(* IEC 61131-3 sources: elnaProjects/ElpcLogic/PomarKc7Unchanged/build_USO_ecl (part 6) *)

  IF NOT onInit THEN

         fb_kran4Close(phaseNumber:=1, act:=_off);
         fb_kran3bOpen(phaseNumber:=2, act:=_on);
              fb_mvOff(phaseNumber:=3, act:=_off);
              fb_pnsOn(phaseNumber:=4, act:=_on);
         fb_kran1Close(phaseNumber:=6, act:=_off);
         fb_kran2Close(phaseNumber:=7, act:=_off);
          fb_kran5Open(phaseNumber:=8, act:=_on);
          fb_autoNuOff(phaseNumber:=9, act:=_reset, waitCompletion:=FALSE);
         fb_autoPnsOff(phaseNumber:=10, act:=_reset, waitCompletion:=FALSE);
        fb_autoAvomOff(phaseNumber:=11, act:=_reset, waitCompletion:=FALSE);
        fb_avom1cmdOff(phaseNumber:=12, act:=_off);
        fb_avom2cmdOff(phaseNumber:=13, act:=_off);
      fb_pInNagLess100(phaseNumber:=14);
           fb_waitKran(phaseNumber:=15, delay:=T#240S);
         fb_pnsWaitOff(phaseNumber:=17, act:=_run, waitCompletion:=TRUE);
             fb_nu1off(phaseNumber:=18, act:=_off);
             fb_nu2off(phaseNumber:=19, act:=_off);
    fb_runUnsuccessful(phaseNumber:=20);

  onInit:=TRUE;
  END_IF;

         fb_kran4Close(StrPh:=kran4Close, Im:=Im.kran4);
         fb_kran3bOpen(StrPh:=kran3bOpen, Im:=Im.kran3b);
              fb_mvOff(StrPh:=mvOff, Im:=Im.mv);
              fb_pnsOn(StrPh:=pnsOn, Im:=Im.pns);

         fb_kran1Close(StrPh:=kran1Close, Im:=Im.kran1);
         fb_kran2Close(StrPh:=kran2Close, Im:=Im.kran2);
          fb_kran5Open(StrPh:=kran5Open, Im:=Im.kran5);
          fb_autoNuOff(StrPh:=autoNuOff, alg:=algoritms.autoNu);
         fb_autoPnsOff(StrPh:=autoPnsOff, alg:=algoritms.autoPns);
        fb_autoAvomOff(StrPh:=autoAvomOff, alg:=algoritms.AutoAvom);
        fb_avom1cmdOff(StrPh:=avom1cmdOff, Im:=Im.v1_Avom);
        fb_avom2cmdOff(StrPh:=avom2cmdOff, Im:=Im.v2_Avom);
      fb_pInNagLess100(StrPh:=pInNagLess100);
           fb_waitKran(StrPh:=waitKran, timer:=AlgTimers.AO_waitKran);
         fb_pnsWaitOff(StrPh:=pnsWaitOff, alg:=algoritms.vibegPNS, waitCompletion:=TRUE);
             fb_nu1off(StrPh:=nu1off, Im:=Im.nu1);
             fb_nu2off(StrPh:=nu2off, Im:=Im.nu2);
    fb_runUnsuccessful(StrPh:=runUnsuccessful);

  StrAlg.CanRun := StrAlg.inCanRun;
  StrAlg.OpcCommandsDisabled := StrAlg.inOpcCommandsDisabled;

  IF StrAlg.isRuning THEN

      StrAlg.hasError := kran4Close.error OR mvOff.error OR pnsOn.error OR kran3bOpen.error
      OR kran1Close.error OR kran2Close.error OR kran5Open.error OR runUnsuccessful.error;

      runPhase(kran4Close);
      runPhase(kran3bOpen);
      runPhase(kran1Close);
      runPhase(kran2Close);
      runPhase(mvOff);

      IF kran1Close.top AND kran2Close.top AND kran4Close.top THEN
          runPhase(kran5Open);
      END_IF;

      IF mvOff.top THEN
            runPhase(autoPnsOff);
      END_IF;

       IF autoPnsOff.top THEN
  	runPhase(pnsOn);
      END_IF;

      IF kran5Open.top THEN
         runPhase(pInNagLess100);
         resetPhase(waitKran);
      END_IF;

     IF pInNagLess100.start AND NOT pInNagLess100.top THEN
  	pInNagLess100.top:=( ai.P_gaza_na_vkhode_nagnetatelia.interval >= _statusAi.NORMAL AND
            ai.P_gaza_na_vkhode_nagnetatelia.value < Ust_Pgaza ) AND
           (ai.P_gaza_na_vykhode_nagnetatelia.interval >= _statusAi.NORMAL AND
            ai.P_gaza_na_vykhode_nagnetatelia.value < Ust_Pgaza);

     END_IF;

      IF pInNagLess100.top AND kran3bOpen.top AND mvOff.top THEN
  	ai.dPmaslo_gaz.Disabled_LA:=TRUE;
            ai.dPmaslo_gaz.Disabled_LW:=TRUE;
            IM.SingleSignals.dP_oilgaz_low.Disabled_Sig:=TRUE;
            resetAiProtection(protections.dP_maslogaz_LA);
            resetDiProtection(protections.dP_masloGaz_LowDI);

            runPhase(autoNuOff);
            runPhase(nu1off);
            runPhase(nu2off);
      END_IF;

       IF nu1off.top AND  nu2off.top THEN
  	runPhase(pnsWaitOff);
      END_IF;

      IF waitKran.top AND (NOT kran5Open.top) THEN
  	runUnsuccessful.error:=TRUE;
      END_IF;

      IF pnsWaitOff.top THEN
  	runPhase(autoAvomOff);
      END_IF;

      IF autoAvomOff.top THEN
  	runPhase(avom1cmdOff);
  	runPhase(avom2cmdOff);
      END_IF;

      IF avom1cmdOff.top AND avom2cmdOff.top THEN
  	 StrAlg.opcCommandsDisabled:=FALSE;
      END_IF;

      StrAlg.isEnded:= avom1cmdOff.top AND avom2cmdOff.top;
  END_IF;

  StrAlg.CanRun := StrAlg.inCanRun;
  StrAlg.OpcCommandsDisabled := StrAlg.inOpcCommandsDisabled;

  (* ---- Если управление с ВУ заблокировано, то  передаем команду из алгоритма ---- *)
  IF StrAlg.inOpcCommandsDisabled THEN
  	StrAlg.inCommand := StrAlg.inCommand_Alg;
  ELSE (* иначе передаем команду с АРМа*)
  	StrAlg.inCommand := StrAlg.inCommand_ARM;
  END_IF;

  _sunpackerCommand(command := StrAlg.inCommand);
  	source := _sunpackerCommand.source;
  	cmd := _sunpackerCommand.cmd;

  IF cmd <> 0 AND lastCmd <> cmd AND (((NOT StrAlg.opcCommandsDisabled) AND source > 0) OR source = 0) then
  	CASE BYTE_TO_INT(cmd) OF
  		(*cmdRun*) 1: 	IF (StrAlg.CanRun) THEN
  					StrAlg.isRuning := TRUE;
  					StrAlg.isEnded := FALSE;
  					StrAlg.hasError := FALSE;
  					(*****************       OnRun       *****************)

                                                    StrAlg.opcCommandsDisabled:=TRUE;
                                                    runIfNotRunningSO(IM.SingleOutputs.IndikicijaAS_fonar);
                                                    runIfNotRunningSO(IM.SingleOutputs.AO_GPA);
                                                    stopPusk(algoritms);
                                                    algManager.nMode:=ModeGpa.MODE_AO;

                                                    runPhase(waitKran);
                                                    runPhase(runUnsuccessful);

                                                    resetDiProtection(protections.mvOff);
                                                    resetAiProtection(protections.Vibratciia_rotora_nagnetatelia_t1_HA);
                                                    resetAiProtection(protections.Vibratciia_rotora_nagnetatelia_t2_HA);
                                                    resetAiProtection(protections.Vibratciia_rotora_nagnetatelia_t3_HA);
                                                    resetAiProtection(protections.Vibratciia_rotora_nagnetatelia_t4_HA);
                                                    resetAiProtection(protections.Vibratciia_STD_t1_HA);
                                                    resetAiProtection(protections.Vibratciia_STD_t2_HA);
                                                    resetDiProtection(protections.Kran1sdvig);
                                                    resetDiProtection(protections.Kran2sdvig);

  					cmd_for_Status := cmd;
  					source_for_Status := source;
  					command_error_for_Status := 0;
  				ELSE
  					StrAlg.isRuning := FALSE;
  					StrAlg.isEnded := FALSE;
  					StrAlg.hasError 	:= FALSE;

  					cmd_for_Status := 0;
  					source_for_Status := source;
  					command_error_for_Status := cmd;
  				END_IF;
  		(*cmdReset*) 2: 	StrAlg.isRuning := FALSE;
  				StrAlg.isEnded := FALSE;
  				StrAlg.hasError 	:= FALSE;

                                           (*****************       OnReset       *****************)
                                          protectManager.inCommand:=PMcommand.RestartAllSignaling;
                                          waitReset(IN:=FALSE);
                                          resetIfRunningSO(IM.SingleOutputs.IndikicijaAS_fonar);
                                          resetIfRunningSO(IM.SingleOutputs.AO_GPA);
                                          resetIfRunning(algoritms.vibegPNS);
                                          algManager.nMode:=ModeGpa.MODE_STOP;
                                          impulseSO(Im.SingleOutputs.SbrosBREO);

                                          resetPhase(kran4Close);
                                          resetPhase(mvOff);
                                          resetPhase(pnsOn);
                                          resetPhase(kran3bOpen);
                                          resetPhase(kran1Close);
                                          resetPhase(kran2Close);
                                          resetPhase(kran5Open);
                                          resetPhase(autoNuOff);
                                          resetPhase(autoPnsOff);
                                          resetPhase(pInNagLess100);
  	                              resetPhase(autoAvomOff);
                                          resetPhase(avom1cmdOff);
                                          resetPhase(avom2cmdOff);
                                          resetPhase(nu1off);
                                          resetPhase(nu2off);
                                          resetPhase(waitKran);
                                          resetPhase(pnsWaitOff);
                                          resetPhase(runUnsuccessful);

  				cmd_for_Status := cmd;
  				source_for_Status := source;
  				command_error_for_Status := 0;
  	END_CASE;
  	resetCmdTimer(IN := false);
  	resetCmdTimerPriznak := TRUE;
  END_IF;
  lastCmd := cmd;

  resetCmdTimer(IN := resetCmdTimerPriznak, PT := T#5S);
  IF resetCmdTimer.Q THEN
  	resetCmdTimerPriznak := FALSE;
  	source_for_Status := 0;
  	cmd_for_Status := 0;
  	command_error_for_Status := 0;
  END_IF;

  StrAlg.Start:= kran4Close.startStatus
              OR mvOff.startStatus
              OR pnsOn.startStatus
              OR kran3bOpen.startStatus
              OR kran1Close.startStatus
              OR kran2Close.startStatus
              OR kran5Open.startStatus
              OR autoNuOff.startStatus
              OR autoPnsOff.startStatus
              OR pInNagLess100.startStatus
              OR autoAvomOff.startStatus
              OR avom1cmdOff.startStatus
              OR avom2cmdOff.startStatus
              OR nu1off.startStatus
              OR nu2off.startStatus
              OR waitKran.startStatus
              OR pnsWaitOff.startStatus
              OR runUnsuccessful.startStatus;

  StrAlg.Error:= kran4Close.errorStatus
              OR mvOff.errorStatus
              OR pnsOn.errorStatus
              OR kran3bOpen.errorStatus
              OR kran1Close.errorStatus
              OR kran2Close.errorStatus
              OR kran5Open.errorStatus
              OR autoNuOff.errorStatus
              OR autoPnsOff.errorStatus
              OR pInNagLess100.errorStatus
              OR autoAvomOff.errorStatus
              OR avom1cmdOff.errorStatus
              OR avom2cmdOff.errorStatus
              OR nu1off.errorStatus
              OR nu2off.errorStatus
              OR waitKran.errorStatus
              OR pnsWaitOff.errorStatus
              OR runUnsuccessful.errorStatus;

  StrAlg.Top:=   kran4Close.topStatus
              OR mvOff.topStatus
              OR pnsOn.topStatus
              OR kran3bOpen.topStatus
              OR kran1Close.topStatus
              OR kran2Close.topStatus
              OR kran5Open.topStatus
              OR autoNuOff.topStatus
              OR autoPnsOff.topStatus
              OR pInNagLess100.topStatus
              OR autoAvomOff.topStatus
              OR avom1cmdOff.topStatus
              OR avom2cmdOff.topStatus
              OR nu1off.topStatus
              OR nu2off.topStatus
              OR waitKran.topStatus
              OR pnsWaitOff.topStatus
              OR runUnsuccessful.topStatus;

  (*TODO: TYPE PROGRAM CODE HERE*)
  StrAlg.status :=  SHL(BYTE_TO_DWORD(source_for_Status), 29)
  			OR SHL(BYTE_TO_DWORD(cmd_for_Status), 26)
  			OR SHL(BYTE_TO_DWORD(command_error_for_Status), 23)
  			OR SHL(BOOL_TO_DWORD(StrAlg.OpcCommandsDisabled ), 21)
  			OR SHL(BOOL_TO_DWORD(StrAlg.hasError),4)
  			OR SHL(BOOL_TO_DWORD(StrAlg.CanRun),2)
  			OR SHL(BOOL_TO_DWORD(StrAlg.isEnded),1)
  			OR BOOL_TO_DWORD(StrAlg.isRuning);
END_FUNCTION_BLOCK

FUNCTION NapryageniaOK : BOOL
  VAR_INPUT
    im : ImConfig;
  END_VAR

  NapryageniaOK:=
  NOT (Im.SingleSignals.NS_G1_G2.Q
  OR Im.SingleSignals.NS_G10_G11.Q
  OR Im.SingleSignals.NS_G13_G14.Q
  OR Im.SingleSignals.NS_G15_G16.Q
  OR Im.SingleSignals.NS_G17.Q
  OR Im.SingleSignals.NS_G18_G19.Q
  OR Im.SingleSignals.NS_G3_G4.Q
  OR Im.SingleSignals.NS_G5_G6.Q
  OR Im.SingleSignals.NS_G7_G8.Q
  OR im.SingleSignals.QF1_on.Q
  OR Im.SingleSignals.QF2_on.Q
  OR Im.SingleSignals.QF23_on.Q
  OR Im.SingleSignals.QF4_QF5_on.Q
  OR Im.SingleSignals.QF6_QF7_on.Q
  OR Im.SingleSignals.QF8_QF9_on.Q
  OR Im.SingleSignals.QF10_QF11_on.Q
  OR im.SingleSignals.QF12_QF13_on.Q
  OR im.SingleSignals.QF22_on.Q
  OR Im.SingleSignals.QF14_QF15_on.Q);
END_FUNCTION

FUNCTION nsCepeiUpravlenya : BOOL
  VAR_INPUT
    im : ImConfig;
  END_VAR

  nsCepeiUpravlenya:=
  	im.kran1.So OR im.kran1.Sz OR
  	im.kran2.So OR im.kran2.Sz OR
  	im.kran4.So OR im.kran4.Sz OR
  	im.kran5.So OR im.kran5.Sz OR
  	(*im.kran6.So OR im.kran6.Sz OR*)
  	im.kran3b.So OR im.kran3b.Sz OR
  	im.pns.breakCmdOn OR
  	im.nu1.breakCmdOn OR
  	im.nu2.breakCmdOn OR
  	im.PNS.breakCmdOn OR
            im.v1_Avom.breakCmdOn OR
            im.v2_Avom.breakCmdOn OR
            (*im.Ten.breakCmdOn OR*)
  	im.mv.breakCmdOff;
END_FUNCTION

FUNCTION discretNS : BOOL
  VAR_INPUT
    di : DiConfig;
  END_VAR

  discretNS:=  ((di.di_0.reliability <> 255)
                OR (di.di_1.reliability <> 255)
                OR (di.di_2.reliability <> 255)
                OR (di.di_3.reliability <> 255)
                OR (di.di_4.reliability <> 255)
                OR (di.di_5.reliability <> 255)
                OR (di.di_6.reliability <> 255)
                OR (di.di_7.reliability <> 255)
                OR (di.di_8.reliability <> 255)
                OR (di.di_9.reliability <> 255)
                OR (di.di_10.reliability <> 255)
                OR (di.di_11.reliability <> 255)
                OR (di.di_12.reliability <> 255)
                OR (di.di_13.reliability <> 255)
                OR (di.di_14.reliability <> 255));
               (* OR (di.di_15.reliability <> 255)); *)
END_FUNCTION

FUNCTION analogsNS : BOOL
  VAR_INPUT
    ai : AiConfig;
  END_VAR
  VAR
    statusAi : TYPE_StatusAi;
  END_VAR

  analogsNS:=
    ((ai.T_obmotki_fazy_1_k.Interval < statusAi.Normal) AND NOT ai.T_obmotki_fazy_1_k.remont)
  OR((ai.T_aktivnogo_zheleza_statora_1_k.Interval < statusAi.Normal) AND NOT ai.T_aktivnogo_zheleza_statora_1_k.remont)
  OR((ai.T_obmotki_fazy_2_k.Interval < statusAi.Normal) AND NOT ai.T_obmotki_fazy_2_k.remont)
  OR((ai.T_aktivnogo_zheleza_statora_2_k.Interval < statusAi.Normal) AND NOT ai.T_aktivnogo_zheleza_statora_2_k.remont)
  OR((ai.T_obmotki_fazy_3_k.Interval < statusAi.Normal) AND NOT ai.T_obmotki_fazy_3_k.remont)
  OR((ai.T_aktivnogo_zheleza_statora_3_k.Interval < statusAi.Normal) AND NOT ai.T_aktivnogo_zheleza_statora_3_k.remont)
  OR((ai.T_masla_v_maslobake.Interval < statusAi.Normal) AND NOT ai.T_masla_v_maslobake.remont)
  OR((ai.T_perednego_opornogo_podshipnika_dvigatelia_t1.Interval < statusAi.Normal) AND NOT ai.T_perednego_opornogo_podshipnika_dvigatelia_t1.remont)
  OR((ai.T_zadnego_opornogo_podshipnika_dvigatelia_t2.Interval < statusAi.Normal) AND NOT ai.T_zadnego_opornogo_podshipnika_dvigatelia_t2.remont)
  OR((ai.T_masla_na_slive_perednego_opornogo_podshipnika_dvigatelia.Interval < statusAi.Normal) AND NOT ai.T_masla_na_slive_perednego_opornogo_podshipnika_dvigatelia.remont)
  OR((ai.T_masla_na_slive_zadnego_opornogo_podshipnika_dvigatelia.Interval < statusAi.Normal) AND NOT ai.T_masla_na_slive_zadnego_opornogo_podshipnika_dvigatelia.remont)
  OR((ai.T_podshipnika_reduktora_t1.Interval < statusAi.Normal) AND NOT ai.T_podshipnika_reduktora_t1.remont)
  OR((ai.T_podshipnika_reduktora_t2.Interval < statusAi.Normal) AND NOT ai.T_podshipnika_reduktora_t2.remont)
  OR((ai.T_podshipnika_reduktora_t3.Interval < statusAi.Normal) AND NOT ai.T_podshipnika_reduktora_t3.remont)
  OR((ai.T_podshipnika_reduktora_t4.Interval < statusAi.Normal) AND NOT ai.T_podshipnika_reduktora_t4.remont)
  OR((ai.T_opornogo_podshipnika_nagnetatelia_t1.Interval < statusAi.Normal) AND NOT ai.T_opornogo_podshipnika_nagnetatelia_t1.remont)
  OR((ai.T_opornogo_podshipnika_nagnetatelia_t2.Interval < statusAi.Normal) AND NOT ai.T_opornogo_podshipnika_nagnetatelia_t2.remont)
  OR((ai.T_opornogo_podshipnika_nagnetatelia_t3.Interval < statusAi.Normal) AND NOT ai.T_opornogo_podshipnika_nagnetatelia_t3.remont)
  OR((ai.T_oporno_upornogo_podshipnika_nagnetatelia_t4.Interval < statusAi.Normal) AND NOT ai.T_oporno_upornogo_podshipnika_nagnetatelia_t4.remont)
  OR((ai.T_masla_do_AVOM.Interval < statusAi.Normal) AND NOT ai.T_masla_do_AVOM.remont)
  OR((ai.T_masla_posle_AVOM.Interval < statusAi.Normal) AND NOT ai.T_masla_posle_AVOM.remont)
  OR((ai.T_gaz_in_nagnetatelia.Interval < statusAi.Normal) AND NOT ai.T_gaz_in_nagnetatelia.remont)
  OR((ai.T_gaz_out_nagnetatelia.Interval < statusAi.Normal) AND NOT ai.T_gaz_out_nagnetatelia.remont)
  OR((ai.T_clodAir_dvigatelia_t1.Interval < statusAi.Normal) AND NOT ai.T_clodAir_dvigatelia_t1.remont)
  OR((ai.T_hotAir_dvigatelia_t1.Interval < statusAi.Normal) AND NOT ai.T_hotAir_dvigatelia_t1.remont)
  OR((ai.dPmaslo_gaz.Interval < statusAi.Normal) AND NOT ai.dPmaslo_gaz.remont)
  OR((ai.dP_gaza_na_konfuzore_nagnetatelia.Interval < statusAi.Normal) AND NOT ai.dP_gaza_na_konfuzore_nagnetatelia.remont)
  OR((ai.P_masla_uplotneniia.Interval < statusAi.Normal) AND NOT ai.P_masla_uplotneniia.remont)
  OR((ai.P_gaza_na_vkhode_nagnetatelia.Interval < statusAi.Normal) AND NOT ai.P_gaza_na_vkhode_nagnetatelia.remont)
  OR((ai.P_gaza_na_vykhode_nagnetatelia.Interval < statusAi.Normal) AND NOT ai.P_gaza_na_vykhode_nagnetatelia.remont)
  OR((ai.P_masla_smazki_nizkoe.Interval < statusAi.Normal) AND NOT ai.P_masla_smazki_nizkoe.remont)
  OR((ai.P_masla_smazki_srednee_posle_nasosov.Interval < statusAi.Normal) AND NOT ai.P_masla_smazki_srednee_posle_nasosov.remont)
  OR((ai.Vibratciia_STD_t1.Interval < statusAi.Normal) AND NOT ai.Vibratciia_STD_t1.remont)
  OR((ai.Vibratciia_STD_t2.Interval < statusAi.Normal) AND NOT ai.Vibratciia_STD_t2.remont)
  OR((ai.Vibratciia_rotora_nagnetatelia_t1.Interval < statusAi.Normal) AND NOT ai.Vibratciia_rotora_nagnetatelia_t1.remont)
  OR((ai.Vibratciia_rotora_nagnetatelia_t2.Interval < statusAi.Normal) AND NOT ai.Vibratciia_rotora_nagnetatelia_t2.remont)
  OR((ai.Vibratciia_rotora_nagnetatelia_t3.Interval < statusAi.Normal) AND NOT ai.Vibratciia_rotora_nagnetatelia_t3.remont)
  OR((ai.Vibratciia_rotora_nagnetatelia_t4.Interval < statusAi.Normal) AND NOT ai.Vibratciia_rotora_nagnetatelia_t4.remont)
  OR((ai.Osevoi_sdvig_rotora_nagnetatelia.Interval < statusAi.Normal) AND NOT ai.Osevoi_sdvig_rotora_nagnetatelia.remont)
  OR((ai.Uroven_masla_v_maslobake.Interval < statusAi.Normal) AND NOT ai.Uroven_masla_v_maslobake.remont)
  OR((ai.Tok_vozbuzhdeniia_vozbuditelia.Interval < statusAi.Normal) AND NOT ai.Tok_vozbuzhdeniia_vozbuditelia.remont)
  OR((ai.Tok_statora_elektrodvigatelia.Interval < statusAi.Normal) AND NOT ai.Tok_statora_elektrodvigatelia.remont)
  OR((ai.Aktivnaia_moshchnost.Interval < statusAi.Normal) AND NOT ai.Aktivnaia_moshchnost.remont)
  OR((ai.Reaktivnaia_moshchnost.Interval < statusAi.Normal) AND NOT ai.Reaktivnaia_moshchnost.remont)
  OR((ai.VoltageSHU_osnovnoi_vvod.Interval < statusAi.Normal) AND NOT ai.VoltageSHU_osnovnoi_vvod.remont)
  OR((ai.VoltageSHU_rezervnyi_vvod.Interval < statusAi.Normal) AND NOT ai.VoltageSHU_rezervnyi_vvod.remont);
END_FUNCTION

FUNCTION nsCepeiControl : BOOL
  VAR_INPUT
    im : ImConfig;
  END_VAR

  nsCepeiControl:= NOT (
  	im.kran1.reliability OR
  	im.kran2.reliability OR
  	im.kran4.reliability OR
  	im.kran5.reliability OR
  	im.kran6.reliability OR
  	im.kran3b.reliability OR
  	im.pns.reliability OR
  	im.nu1.reliability OR
  	im.nu2.reliability OR
  	im.PNS.reliability OR
            im.v1_Avom.reliability OR
            im.v2_Avom.reliability OR
            im.Ten.reliability OR
  	im.mv.reliability);
END_FUNCTION

FUNCTION_BLOCK ppuAlg
  VAR_IN_OUT
    StrAlg : struct_Alg;
  END_VAR
  VAR
    Sau_ok : struct_PhaseAlgoritm;
    Voltage_ok : struct_PhaseAlgoritm;
    controlCircuits_ok : struct_PhaseAlgoritm;
    controlCircuitsIM_ok : struct_PhaseAlgoritm;
  END_VAR
  VAR_IN_OUT
    BEAO_otKnSHU : struct_PhaseAlgoritm;
    circuitAO_ok : struct_PhaseAlgoritm;
    BREO_Srabotal : struct_PhaseAlgoritm;
    DI_ok : struct_PhaseAlgoritm;
    AI_ok : struct_PhaseAlgoritm;
    Loil_ok : struct_PhaseAlgoritm;
    Toil_ok : struct_PhaseAlgoritm;
    mvOff : struct_PhaseAlgoritm;
    Kr_1_close : struct_PhaseAlgoritm;
    Kr_2_close : struct_PhaseAlgoritm;
    Kr_3b_open : struct_PhaseAlgoritm;
    Kr_4_close : struct_PhaseAlgoritm;
    Kr_5_open : struct_PhaseAlgoritm;
    PNS_off : struct_PhaseAlgoritm;
    NU_1_off : struct_PhaseAlgoritm;
    NU_2_off : struct_PhaseAlgoritm;
    Avom_1_off : struct_PhaseAlgoritm;
    Avom_2_off : struct_PhaseAlgoritm;
    Est_rezerv_NU : struct_PhaseAlgoritm;
    Not_AO_NO_EAO : struct_PhaseAlgoritm;
    Not_AS_PS : struct_PhaseAlgoritm;
    BusketTest : struct_PhaseAlgoritm;
    BusketRolledIn : struct_PhaseAlgoritm;
  END_VAR
  VAR
    fb_Sau_ok : fb_ph_CustomPhase;
    fb_Voltage_ok : fb_ph_CustomPhase;
    fb_controlCircuits_ok : fb_ph_CustomPhase;
    fb_controlCircuitsIM_ok : fb_ph_CustomPhase;
    fb_BEAO_otKnSHU : fb_ph_CustomPhase;
    fb_circuitAO_ok : fb_ph_CustomPhase;
    fb_BREO_Srabotal : fb_ph_CustomPhase;
    fb_DI_ok : fb_ph_CustomPhase;
    fb_AI_ok : fb_ph_CustomPhase;
    fb_Loil_ok : fb_ph_CustomPhase;
    fb_Toil_ok : fb_ph_CustomPhase;
    fb_mvOff : fb_ph_CustomPhase;
    fb_Kr_1_close : fb_ph_CustomPhase;
    fb_Kr_2_close : fb_ph_CustomPhase;
    fb_Kr_3b_open : fb_ph_CustomPhase;
    fb_Kr_4_close : fb_ph_CustomPhase;
    fb_Kr_5_open : fb_ph_CustomPhase;
    fb_PNS_off : fb_ph_CustomPhase;
    fb_NU_1_off : fb_ph_CustomPhase;
    fb_NU_2_off : fb_ph_CustomPhase;
    fb_Avom_1_off : fb_ph_CustomPhase;
    fb_Avom_2_off : fb_ph_CustomPhase;
    fb_Est_rezerv_NU : fb_ph_CustomPhase;
    fb_Not_AO_NO_EAO : fb_ph_CustomPhase;
    fb_Not_AS_PS : fb_ph_CustomPhase;
    fb_BusketTest : fb_ph_CustomPhase;
    fb_BusketRolledIn : fb_ph_CustomPhase;
    _sunpackerCommand : fb_sunpackerCommand;
    modeR_Trig : R_TRIG;
    modeF_Trig : F_TRIG;
    _statusAi : TYPE_StatusAi;
    _Answers : TYPE_Answers;
    _statusDualInput : TYPE_statusDualInput;
    _DualStateImAction : TYPE_DualStateImAction;
    _PhaseAlgoritmAction : TYPE_PhaseAlgoritmAction;
    _basketStats : TYPE_basketStats;
  END_VAR
  VAR_OUTPUT
    puskAllowed : BOOL;
    testAllowed : BOOL;
  END_VAR
  VAR
    ppuDone : BOOL;
    source : BYTE;
    cmd : BYTE;
    lastCmd : BYTE;
    source_for_Status : BYTE;
    cmd_for_Status : BYTE;
    command_error_for_Status : BYTE;
    resetCmdTimer : TON;
    resetCmdTimerPriznak : BOOL;
    onInit : BOOL;
  END_VAR
  VAR_EXTERNAL
    IM : ImConfig;
    ai : AiConfig;
    di : DiConfig;
    algManager : struct_AlgoritmsManager;
    protectManager : struct_ProtectionsManager;
    NotHasRezervNU : BOOL;
    ModeGpa : TYPE_ModeGpa;
    algoritms : AlgoritmsConfig;
  END_VAR

  IF NOT onInit THEN
                fb_Sau_ok(phaseNumber:=0);
            fb_Voltage_ok(phaseNumber:=1);
    fb_controlCircuits_ok(phaseNumber:=2);
  fb_controlCircuitsIM_ok(phaseNumber:=5);
          fb_BEAO_otKnSHU(phaseNumber:=6);
          fb_circuitAO_ok(phaseNumber:=7);
         fb_BREO_Srabotal(phaseNumber:=9);
                 fb_DI_ok(phaseNumber:=10);
                 fb_AI_ok(phaseNumber:=11);
               fb_Loil_ok(phaseNumber:=12);
               fb_Toil_ok(phaseNumber:=13);
                 fb_mvOff(phaseNumber:=14);
            fb_Kr_1_close(phaseNumber:=15);
            fb_Kr_2_close(phaseNumber:=16);
            fb_Kr_3b_open(phaseNumber:=17);
            fb_Kr_4_close(phaseNumber:=18);
             fb_Kr_5_open(phaseNumber:=19);
               fb_PNS_off(phaseNumber:=20);
              fb_NU_1_off(phaseNumber:=21);
              fb_NU_2_off(phaseNumber:=22);
            fb_Avom_1_off(phaseNumber:=23);
            fb_Avom_2_off(phaseNumber:=24);
         fb_Est_rezerv_NU(phaseNumber:=25);
         fb_Not_AO_NO_EAO(phaseNumber:=26);
             fb_Not_AS_PS(phaseNumber:=27);
            fb_BusketTest(phaseNumber:=28);
        fb_BusketRolledIn(phaseNumber:=29);

  onInit:=TRUE;
  END_IF;

                fb_Sau_ok(StrPh:=Sau_ok);
            fb_Voltage_ok(StrPh:=Voltage_ok);
    fb_controlCircuits_ok(StrPh:=controlCircuits_ok);
  fb_controlCircuitsIM_ok(StrPh:=controlCircuitsIM_ok);
          fb_BEAO_otKnSHU(StrPh:=BEAO_otKnSHU);
          fb_circuitAO_ok(StrPh:=circuitAO_ok);
         fb_BREO_Srabotal(StrPh:=BREO_Srabotal);
                 fb_DI_ok(StrPh:=DI_ok);
                 fb_AI_ok(StrPh:=AI_ok);
               fb_Loil_ok(StrPh:=Loil_ok);
               fb_Toil_ok(StrPh:=Toil_ok);
                 fb_mvOff(StrPh:=mvOff);
            fb_Kr_1_close(StrPh:=Kr_1_close);
            fb_Kr_2_close(StrPh:=Kr_2_close);
            fb_Kr_3b_open(StrPh:=Kr_3b_open);
            fb_Kr_4_close(StrPh:=Kr_4_close);
             fb_Kr_5_open(StrPh:=Kr_5_open);
               fb_PNS_off(StrPh:=PNS_off);
              fb_NU_1_off(StrPh:=NU_1_off);
              fb_NU_2_off(StrPh:=NU_2_off);
            fb_Avom_1_off(StrPh:=Avom_1_off);
            fb_Avom_2_off(StrPh:=Avom_2_off);
         fb_Est_rezerv_NU(StrPh:=Est_rezerv_NU);
         fb_Not_AO_NO_EAO(StrPh:=Not_AO_NO_EAO);
             fb_Not_AS_PS(StrPh:=Not_AS_PS);
            fb_BusketTest(StrPh:=BusketTest);
        fb_BusketRolledIn(StrPh:=BusketRolledIn);

  IF StrAlg.isRuning THEN

      Sau_ok.top:= (*(NOT kontroller.diagnostic.ns)  OR kontroller.imit;*) TRUE;
      Voltage_ok.top	:=NapryageniaOK(IM);
      controlCircuits_ok.top	:=NOT nsCepeiUpravlenya(IM);
      controlCircuitsIM_ok.top	:=NOT nsCepeiControl(IM);
      BEAO_otKnSHU.top	:=NOT Im.singleSignals.BEO_ON_knopkaSHU.Q AND Im.singleSignals.BEO_ON_knopkaSHU.reliability;
      circuitAO_ok.top	:=NOT Im.singleSignals.AO_KC.Q AND Im.singleSignals.AO_KC.reliability;
      BREO_Srabotal.top	:=NOT Im.singleSignals.BEO_Srabat.Q AND Im.singleSignals.BEO_Srabat.reliability;
      DI_ok.top	:=NOT discretNS(di);
      AI_ok.top	:=NOT analogsNS(ai);
      mvOff.top:=Im.mv.onStatus = _statusDualInput.STATUS_OFF;
      Toil_ok.top:=(ai.T_masla_v_maslobake.interval = _statusAi.normal);
      Loil_ok.top:=(ai.Uroven_masla_v_maslobake.interval= _statusAi.normal) ;

      Kr_1_close.top:=Im.kran1.onStatus = _statusDualInput.STATUS_OFF;
      Kr_2_close.top:=Im.kran2.onStatus = _statusDualInput.STATUS_OFF;
      Kr_3b_open.top:=Im.kran3b.onStatus = _statusDualInput.STATUS_ON;
      Kr_4_close.top:=Im.kran4.onStatus = _statusDualInput.STATUS_OFF;
      Kr_5_open.top:=	Im.kran5.onStatus = _statusDualInput.STATUS_ON;
      PNS_off.top:=	Im.pns.onStatus = _statusDualInput.STATUS_OFF;
      NU_1_off.top:=	Im.nu1.onStatus = _statusDualInput.STATUS_OFF;
      NU_2_off.top:=	Im.nu2.onStatus = _statusDualInput.STATUS_OFF;
      Avom_1_off.top:=Im.v1_Avom.onStatus = _statusDualInput.STATUS_OFF;
      Avom_2_off.top:=Im.v2_Avom.onStatus = _statusDualInput.STATUS_OFF;

      Est_rezerv_NU.top:= NOT NotHasRezervNU;
      Not_AO_NO_EAO.top:=	   NOT ( Im.singleOutputs.AO_GPA.q
                                      OR Im.singleSignals.AO_KC.q
                                      OR Im.singleSignals.AOGPA_knopkaSHU.q
                                      OR Im.singleSignals.AOGPA_PRU.q
                                      OR Im.singleSignals.NOGPA_knopkaSHU.q
                                      OR Im.singleSignals.BEO_Srabat.q);

      Not_AS_PS.top:=	NOT (algManager.DiscretPS OR algManager.analogsPS OR algManager.ProtectionSignaling);
      BusketTest.top:=Im.mv.basketStatus = _basketStats.BASKET_ROLLEDOUT;
      BusketRolledIn.top:=Im.mv.basketStatus = _basketStats.BASKET_RolledIN;

      ppuDone:=                 Sau_ok.top AND
  			Voltage_ok.top AND
  			controlCircuits_ok.top AND
  			controlCircuitsIM_ok.top AND
  			circuitAO_ok.top AND
  			BEAO_otKnSHU.top	AND
  			BREO_Srabotal.top	AND
  			DI_ok.top AND
  			AI_ok.top AND
  			Loil_ok.top AND
  			Toil_ok.top AND
  			mvOff.top AND
  			Kr_1_close.top AND
  			Kr_2_close.top AND
  			Kr_3b_open.top AND
  			Kr_4_close.top AND
  			Kr_5_open.top AND
  			PNS_off.top AND
  			NU_1_off.top AND
  			NU_2_off.top AND
  			Avom_1_off.top AND
  			Avom_2_off.top AND
  			Est_rezerv_NU.top AND
  			Not_AO_NO_EAO.top AND
  			Not_AS_PS.top ;

      puskAllowed:= ppuDone AND Im.mv.basketStatus = _basketStats.BASKET_ROLLEDIN;
      testAllowed:= ppuDone AND Im.mv.basketStatus = _basketStats.BASKET_ROLLEDOUT;

      modeR_Trig(CLK:=puskAllowed);
      modeF_Trig(CLK:=puskAllowed);

      IF modeR_Trig.Q THEN
  	algManager.nMode:= ModeGpa.MODE_READY;
      END_IF;
      IF modeF_Trig.Q THEN
  	algManager.nMode:= ModeGpa.MODE_STOP;
      END_IF;

      IF puskAllowed THEN
          algoritms.Apusk.inCanRun:= TRUE;
          algoritms.SemiAutoPusk.inCanRun:= TRUE;
      ELSE
          algoritms.Apusk.inCanRun:= FALSE;
          algoritms.SemiAutoPusk.inCanRun:= FALSE;
      END_IF;

      IF testAllowed THEN
          algoritms.testPms.inCanRun:=  TRUE;
          algoritms.testdPmg.inCanRun:= TRUE;
          algoritms.puskK.inCanRun:=    TRUE;
          algoritms.puskV.inCanRun:=    TRUE;
      ELSE
          algoritms.testPms.inCanRun:=  FALSE;
          algoritms.testdPmg.inCanRun:= FALSE;
          algoritms.puskK.inCanRun:=    FALSE;
          algoritms.puskV.inCanRun:=    FALSE;
      END_IF;

  END_IF;

  StrAlg.CanRun := StrAlg.inCanRun;
  StrAlg.OpcCommandsDisabled := StrAlg.inOpcCommandsDisabled;

  (* ---- Если управление с ВУ заблокировано, то  передаем команду из алгоритма ---- *)
  IF StrAlg.inOpcCommandsDisabled THEN
  	StrAlg.inCommand := StrAlg.inCommand_Alg;
  ELSE (* иначе передаем команду с АРМа*)
  	StrAlg.inCommand := StrAlg.inCommand_ARM;
  END_IF;

  _sunpackerCommand(command := StrAlg.inCommand);
  	source := _sunpackerCommand.source;
  	cmd := _sunpackerCommand.cmd;

  IF cmd <> 0 AND lastCmd <> cmd AND (((NOT StrAlg.opcCommandsDisabled) AND source > 0) OR source = 0) then
  	CASE BYTE_TO_INT(cmd) OF
  		(*cmdRun*) 1: 	IF (StrAlg.CanRun) THEN
  					StrAlg.isRuning := TRUE;
  					StrAlg.isEnded := FALSE;
  					StrAlg.hasError := FALSE;
  					(*****************       OnRun       *****************)

  					cmd_for_Status := cmd;
  					source_for_Status := source;
  					command_error_for_Status := 0;
  				ELSE
  					StrAlg.isRuning := FALSE;
  					StrAlg.isEnded := FALSE;
  					StrAlg.hasError 	:= FALSE;

  					cmd_for_Status := 0;
  					source_for_Status := source;
  					command_error_for_Status := cmd;
  				END_IF;
  		(*cmdReset*) 2: 	StrAlg.isRuning := FALSE;
  				StrAlg.isEnded := FALSE;
  				StrAlg.hasError 	:= FALSE;

                                           (*****************       OnReset       *****************)

                                                    resetPhase(Sau_ok);
                                                    resetPhase(Voltage_ok);
                                                    resetPhase(controlCircuits_ok);
                                                    resetPhase(controlCircuitsIM_ok);
                                                    resetPhase(BEAO_otKnSHU);
                                                    resetPhase(circuitAO_ok);
                                                    resetPhase(BREO_Srabotal);
                                                    resetPhase(DI_ok);
                                                    resetPhase(AI_ok);
                                                    resetPhase(Loil_ok);
                                                    resetPhase(Toil_ok);
                                                    resetPhase(mvOff);
                                                    resetPhase(Kr_1_close);
                                                    resetPhase(Kr_2_close);
                                                    resetPhase(Kr_3b_open);
                                                    resetPhase(Kr_4_close);
                                                    resetPhase(Kr_5_open);
                                                    resetPhase(PNS_off);
                                                    resetPhase(NU_1_off);
                                                    resetPhase(NU_2_off);
                                                    resetPhase(Avom_1_off);
                                                    resetPhase(Avom_2_off);
                                                    resetPhase(Est_rezerv_NU);
                                                    resetPhase(Not_AO_NO_EAO);
                                                    resetPhase(Not_AS_PS);
                                                    resetPhase(BusketTest);
                                                    resetPhase(BusketRolledIn);

                                                    algoritms.testPms.inCanRun:=  FALSE;
                                                    algoritms.testdPmg.inCanRun:= FALSE;
                                                    algoritms.puskK.inCanRun:=    FALSE;
                                                    algoritms.puskV.inCanRun:=    FALSE;

                                          StrAlg.inCanRun:=FALSE;
                                          puskAllowed:=FALSE;
                                          testAllowed:=FALSE;
                                          modeR_Trig(CLK:=FALSE);
                                          modeF_Trig(CLK:=FALSE);

  				cmd_for_Status := cmd;
  				source_for_Status := source;
  				command_error_for_Status := 0;
  	END_CASE;
  	resetCmdTimer(IN := false);
  	resetCmdTimerPriznak := TRUE;
  END_IF;
  lastCmd := cmd;

  resetCmdTimer(IN := resetCmdTimerPriznak, PT := T#5S);
  IF resetCmdTimer.Q THEN
  	resetCmdTimerPriznak := FALSE;
  	source_for_Status := 0;
  	cmd_for_Status := 0;
  	command_error_for_Status := 0;
  END_IF;

  StrAlg.Start:= Sau_ok.startStatus
              OR Voltage_ok.startStatus
              OR controlCircuits_ok.startStatus
              OR controlCircuitsIM_ok.startStatus
              OR BEAO_otKnSHU.startStatus
              OR circuitAO_ok.startStatus
              OR BREO_Srabotal.startStatus
              OR DI_ok.startStatus
              OR AI_ok.startStatus
              OR Loil_ok.startStatus
              OR Toil_ok.startStatus
              OR mvOff.startStatus
              OR Kr_1_close.startStatus
              OR Kr_2_close.startStatus
              OR Kr_3b_open.startStatus
              OR Kr_4_close.startStatus
              OR Kr_5_open.startStatus
              OR PNS_off.startStatus
              OR NU_1_off.startStatus
              OR NU_2_off.startStatus
              OR Avom_1_off.startStatus
              OR Avom_2_off.startStatus
              OR Est_rezerv_NU.startStatus
              OR Not_AO_NO_EAO.startStatus
              OR Not_AS_PS.startStatus
              OR BusketTest.startStatus
              OR BusketRolledIn.startStatus;

  StrAlg.Error:= Sau_ok.errorStatus
              OR Voltage_ok.errorStatus
              OR controlCircuits_ok.errorStatus
              OR controlCircuitsIM_ok.errorStatus
              OR BEAO_otKnSHU.errorStatus
              OR circuitAO_ok.errorStatus
              OR BREO_Srabotal.errorStatus
              OR DI_ok.errorStatus
              OR AI_ok.errorStatus
              OR Loil_ok.errorStatus
              OR Toil_ok.errorStatus
              OR mvOff.errorStatus
              OR Kr_1_close.errorStatus
              OR Kr_2_close.errorStatus
              OR Kr_3b_open.errorStatus
              OR Kr_4_close.errorStatus
              OR Kr_5_open.errorStatus
              OR PNS_off.errorStatus
              OR NU_1_off.errorStatus
              OR NU_2_off.errorStatus
              OR Avom_1_off.errorStatus
              OR Avom_2_off.errorStatus
              OR Est_rezerv_NU.errorStatus
              OR Not_AO_NO_EAO.errorStatus
              OR Not_AS_PS.errorStatus
              OR BusketTest.errorStatus
              OR BusketRolledIn.errorStatus;

  StrAlg.Top:=   Sau_ok.topStatus
              OR Voltage_ok.topStatus
              OR controlCircuits_ok.topStatus
              OR controlCircuitsIM_ok.topStatus
              OR BEAO_otKnSHU.topStatus
              OR circuitAO_ok.topStatus
              OR BREO_Srabotal.topStatus
              OR DI_ok.topStatus
              OR AI_ok.topStatus
              OR Loil_ok.topStatus
              OR Toil_ok.topStatus
              OR mvOff.topStatus
              OR Kr_1_close.topStatus
              OR Kr_2_close.topStatus
              OR Kr_3b_open.topStatus
              OR Kr_4_close.topStatus
              OR Kr_5_open.topStatus
              OR PNS_off.topStatus
              OR NU_1_off.topStatus
              OR NU_2_off.topStatus
              OR Avom_1_off.topStatus
              OR Avom_2_off.topStatus
              OR Est_rezerv_NU.topStatus
              OR Not_AO_NO_EAO.topStatus
              OR Not_AS_PS.topStatus
              OR BusketTest.topStatus
              OR BusketRolledIn.topStatus;

  (*TODO: TYPE PROGRAM CODE HERE*)
  StrAlg.status :=  SHL(BYTE_TO_DWORD(source_for_Status), 29)
  			OR SHL(BYTE_TO_DWORD(cmd_for_Status), 26)
  			OR SHL(BYTE_TO_DWORD(command_error_for_Status), 23)
  			OR SHL(BOOL_TO_DWORD(StrAlg.OpcCommandsDisabled ), 21)
                                OR SHL(BOOL_TO_DWORD(testAllowed),16)
                                OR SHL(BOOL_TO_DWORD(puskAllowed),15)
  			OR SHL(BOOL_TO_DWORD(StrAlg.hasError),4)
  			OR SHL(BOOL_TO_DWORD(StrAlg.CanRun),2)
  			OR SHL(BOOL_TO_DWORD(StrAlg.isEnded),1)
  			OR BOOL_TO_DWORD(StrAlg.isRuning);
END_FUNCTION_BLOCK

FUNCTION_BLOCK fb_ph_DIprotection
  VAR_IN_OUT
    StrDiP : struct_DiProtection;
  END_VAR
  VAR_INPUT
    act : TYPE_PhaseAlgoritmAction;
    PhaseNumber : UINT;
  END_VAR
  VAR_IN_OUT
    StrPh : struct_PhaseAlgoritm;
  END_VAR
  VAR
    CommandFault_Trig : R_TRIG;
    reset_Trig : R_TRIG;
    _statusDualInput : TYPE_statusDualInput;
  END_VAR

  IF StrPh.run AND NOT StrPh.start THEN
  	StrPh.start := TRUE;
  	StrPh.top := FALSE;
  	StrPh.error := FALSE;
            StrPh.run:=FALSE;

  	CASE act OF
  		(*PhaseAlgoritmAction.run*)    _run : runDiProtection(StrDiP); (*cmd_run*)
  		(*PhaseAlgoritmAction.reset*)_reset : resetDiProtection(StrDiP); (*cmd_reset*)
  	END_CASE;
  END_IF;

  IF StrPh.start AND NOT StrPh.top THEN
                      CommandFault_Trig(CLK := StrDiP.hasError);
                      IF CommandFault_Trig.Q THEN
  	          StrPh.error := TRUE;
                      END_IF;

  		CASE act OF
  		(*PhaseAlgoritmAction.run*)    _run:    StrPh.top:=StrDiP.isRunning;

  		(*PhaseAlgoritmAction.reset*) _reset:   StrPh.top := NOT StrDiP.isRunning;
  		END_CASE;

  END_IF;

  IF StrPh.top THEN
  StrPh.error := FALSE;
  END_IF;

  reset_Trig(CLK := StrPh.reset);
  IF reset_Trig.Q THEN
            StrPh.start := FALSE;
  	StrPh.error := FALSE;
  	StrPh.top := FALSE;
            StrPh.run:=FALSE;
            StrPh.reset:=FALSE;
  END_IF;

  StrPh.startStatus := SHL(BOOL_TO_DWORD(StrPh.start), PhaseNumber);
  StrPh.errorStatus := SHL(BOOL_TO_DWORD(StrPh.error), PhaseNumber);
  StrPh.topStatus := SHL(BOOL_TO_DWORD(StrPh.top), PhaseNumber);
END_FUNCTION_BLOCK

FUNCTION_BLOCK fillingAlg
  VAR_IN_OUT
    StrAlg : struct_Alg;
  END_VAR
  VAR
    BreakPuskTimer : struct_PhaseAlgoritm;
    kran3bOpen : struct_PhaseAlgoritm;
    kran4Open : struct_PhaseAlgoritm;
    waitAfterKran4 : struct_PhaseAlgoritm;
    kran5Close : struct_PhaseAlgoritm;
    didPKran1 : struct_PhaseAlgoritm;
    kran1Open : struct_PhaseAlgoritm;
    kran2Open : struct_PhaseAlgoritm;
    kran3bClose : struct_PhaseAlgoritm;
    kran4Close : struct_PhaseAlgoritm;
    RunProtection_kr1 : struct_PhaseAlgoritm;
    RunProtection_kr2 : struct_PhaseAlgoritm;
    waitAfterKran5 : struct_PhaseAlgoritm;
    testUnsuccessfulFilling : struct_PhaseAlgoritm;
    fb_BreakPuskTimer : fb_ph_Timer;
    fb_kran3bOpen : fb_ph_Kran;
    fb_kran4Open : fb_ph_Kran;
    fb_waitAfterKran4 : fb_ph_Timer;
    fb_kran5Close : fb_ph_Kran;
    fb_didPKran1 : fb_ph_CustomPhase;
    fb_kran1Open : fb_ph_Kran;
    fb_kran2Open : fb_ph_Kran;
    fb_kran3bClose : fb_ph_Kran;
    fb_kran4Close : fb_ph_Kran;
    fb_RunProtection_kr1 : fb_ph_DIprotection;
    fb_RunProtection_kr2 : fb_ph_DIprotection;
    fb_waitAfterKran5 : fb_ph_Timer;
    fb_testUnsuccessfulFilling : fb_ph_CustomPhase;
    _sunpackerCommand : fb_sunpackerCommand;
    _DualStateImAction : TYPE_DualStateImAction;
    _PhaseAlgoritmAction : TYPE_PhaseAlgoritmAction;
    source : BYTE;
    cmd : BYTE;
    lastCmd : BYTE;
    source_for_Status : BYTE;
    cmd_for_Status : BYTE;
    command_error_for_Status : BYTE;
    resetCmdTimer : TON;
    resetCmdTimerPriznak : BOOL;
    onInit : BOOL;
    waitReset : TON;
  END_VAR
  VAR_EXTERNAL
    IM : ImConfig;
    ai : AiConfig;
    protections : ProtectionsConfig;
    AlgTimers : struct_AlgTimers;
    algoritms : AlgoritmsConfig;
  END_VAR

  IF NOT onInit THEN

           fb_BreakPuskTimer(phaseNumber:=0, delay:=T#240S);
               fb_kran3bOpen(phaseNumber:=1, act:=_on);
                fb_kran4Open(phaseNumber:=2, act:=_on);
           fb_waitAfterKran4(phaseNumber:=3, delay:=T#10S);
               fb_kran5Close(phaseNumber:=4, act:=_off);
                fb_didPKran1(phaseNumber:=5);
                fb_kran1Open(phaseNumber:=7, act:=_on);
                fb_kran2Open(phaseNumber:=8, act:=_on);
              fb_kran3bClose(phaseNumber:=9, act:=_off);
               fb_kran4Close(phaseNumber:=10, act:=_off);
        fb_RunProtection_kr1(phaseNumber:=11, act:=_run);
        fb_RunProtection_kr2(phaseNumber:=12, act:=_run);
           fb_waitAfterKran5(phaseNumber:=13, delay:=T#60S);
  fb_testUnsuccessfulFilling(phaseNumber:=17);

  onInit:=TRUE;
  END_IF;

           fb_BreakPuskTimer(StrPh:=BreakPuskTimer, timer:=AlgTimers.filling_BreakPuskTimer);
               fb_kran3bOpen(StrPh:=kran3bOpen, Im:=Im.kran3b);
                fb_kran4Open(StrPh:=kran4Open, Im:=Im.kran4);
           fb_waitAfterKran4(StrPh:=waitAfterKran4, timer:=AlgTimers.filling_waitAfterKran4);
               fb_kran5Close(StrPh:=kran5Close, Im:=Im.kran5);
                fb_didPKran1(StrPh:=didPKran1);
                fb_kran1Open(StrPh:=kran1Open, Im:=Im.kran1);
                fb_kran2Open(StrPh:=kran2Open, Im:=Im.kran2);
              fb_kran3bClose(StrPh:=kran3bClose, Im:=Im.kran3b);
               fb_kran4Close(StrPh:=kran4Close, Im:=Im.kran4);
        fb_RunProtection_kr1(StrPh:=RunProtection_kr1 , StrDiP:=protections.Kran1sdvig);
        fb_RunProtection_kr2(StrPh:=RunProtection_kr2 , StrDiP:=protections.Kran2sdvig);
           fb_waitAfterKran5(StrPh:=waitAfterKran5, timer:=AlgTimers.filling_waitAfterKran5);
  fb_testUnsuccessfulFilling(StrPh:=testUnsuccessfulFilling);

  StrAlg.CanRun := StrAlg.inCanRun;
  StrAlg.OpcCommandsDisabled := StrAlg.inOpcCommandsDisabled;

  IF StrAlg.isRuning THEN

      StrAlg.hasError := kran3bOpen.error OR kran4Open.error OR kran5Close.error OR kran5Close.error
      OR kran1Open.error OR kran2Open.error OR kran3bClose.error OR kran4Close.error OR testUnsuccessfulFilling.error;

      IF kran4Open.top THEN
          runPhase(waitAfterKran4);
      END_IF;

      IF waitAfterKran4.top THEN
          runPhase(kran5Close);
      END_IF;

      IF kran3bOpen.top AND kran5Close.top THEN
         runPhase(waitAfterKran5);
         runPhase(didPKran1);
      END_IF;

      IF didPKran1.start AND NOT didPKran1.top THEN
      didPKran1.top:= im.singleSignals.dP_gazgaz_Kran1.Q;
      END_IF;

      IF waitAfterKran5.top AND didPKran1.top THEN
            runPhase(kran1Open);
  	runPhase(kran2Open);
      END_IF;

      IF kran1Open.top AND kran2Open.top THEN
            runPhase(kran4Close);
  	runPhase(kran3bClose);
      END_IF;

      IF kran4Close.top AND kran3bClose.top THEN

            runPhase(RunProtection_kr1);
            runPhase(RunProtection_kr2);

            runAiProtection(protections.Vibratciia_STD_t1_HA);
            runAiProtection(protections.Vibratciia_STD_t1_HA);
            runAiProtection(protections.Vibratciia_rotora_nagnetatelia_t1_HA);
            runAiProtection(protections.Vibratciia_rotora_nagnetatelia_t2_HA);
            runAiProtection(protections.Vibratciia_rotora_nagnetatelia_t3_HA);
            runAiProtection(protections.Vibratciia_rotora_nagnetatelia_t4_HA);

      END_IF;

      IF BreakPuskTimer.top AND NOT (RunProtection_kr1.top AND RunProtection_kr2.top ) THEN
  	testUnsuccessfulFilling.error:=TRUE;
      END_IF;

      IF RunProtection_kr1.top AND RunProtection_kr2.top THEN
            resetPhase(BreakPuskTimer);
  	waitReset(IN:=TRUE, PT:= T#2S);
      END_IF;

      IF waitReset.Q AND NOT (algoritms.Apusk.isRuning OR algoritms.SemiAutoPusk.isRuning) THEN
  	resetIfRunning(StrAlg);
      END_IF;

      StrAlg.isEnded:= RunProtection_kr1.top AND RunProtection_kr2.top;
  END_IF;

  StrAlg.CanRun := StrAlg.inCanRun;
  StrAlg.OpcCommandsDisabled := StrAlg.inOpcCommandsDisabled;

  (* ---- Если управление с ВУ заблокировано, то  передаем команду из алгоритма ---- *)
  IF StrAlg.inOpcCommandsDisabled THEN
  	StrAlg.inCommand := StrAlg.inCommand_Alg;
  ELSE (* иначе передаем команду с АРМа*)
  	StrAlg.inCommand := StrAlg.inCommand_ARM;
  END_IF;

  _sunpackerCommand(command := StrAlg.inCommand);
  	source := _sunpackerCommand.source;
  	cmd := _sunpackerCommand.cmd;

  IF cmd <> 0 AND lastCmd <> cmd AND (((NOT StrAlg.opcCommandsDisabled) AND source > 0) OR source = 0) then
  	CASE BYTE_TO_INT(cmd) OF
  		(*cmdRun*) 1: 	IF (StrAlg.CanRun) THEN
  					StrAlg.isRuning := TRUE;
  					StrAlg.isEnded := FALSE;
  					StrAlg.hasError := FALSE;
  					(*****************       OnRun       *****************)

                                                    runPhase(kran3bOpen);
                                                    runPhase(kran4Open);
                                                    runPhase(BreakPuskTimer);
                                                    runPhase(testUnsuccessfulFilling);

  					cmd_for_Status := cmd;
  					source_for_Status := source;
  					command_error_for_Status := 0;
  				ELSE
  					StrAlg.isRuning := FALSE;
  					StrAlg.isEnded := FALSE;
  					StrAlg.hasError 	:= FALSE;

  					cmd_for_Status := 0;
  					source_for_Status := source;
  					command_error_for_Status := cmd;
  				END_IF;
  		(*cmdReset*) 2: 	StrAlg.isRuning := FALSE;
  				StrAlg.isEnded := FALSE;
  				StrAlg.hasError 	:= FALSE;

                                           (*****************       OnReset       *****************)
                                          StrAlg.inCanRun:=FALSE;
                                          waitReset(IN:=FALSE);

                                          resetPhase(BreakPuskTimer);
                                          resetPhase(kran3bOpen);
                                          resetPhase(kran4Open);
                                          resetPhase(waitAfterKran4);
                                          resetPhase(kran5Close);
                                          resetPhase(didPKran1);
                                          resetPhase(kran1Open);
                                          resetPhase(kran2Open);
                                          resetPhase(kran3bClose);
                                          resetPhase(kran4Close);
  	                              resetPhase(RunProtection_kr1);
                                          resetPhase(RunProtection_kr2);
                                          resetPhase(waitAfterKran5);
                                          resetPhase(testUnsuccessfulFilling);

  				cmd_for_Status := cmd;
  				source_for_Status := source;
  				command_error_for_Status := 0;
  	END_CASE;
  	resetCmdTimer(IN := false);
  	resetCmdTimerPriznak := TRUE;
  END_IF;
  lastCmd := cmd;

  resetCmdTimer(IN := resetCmdTimerPriznak, PT := T#5S);
  IF resetCmdTimer.Q THEN
  	resetCmdTimerPriznak := FALSE;
  	source_for_Status := 0;
  	cmd_for_Status := 0;
  	command_error_for_Status := 0;
  END_IF;

  StrAlg.Start:= BreakPuskTimer.startStatus
              OR kran3bOpen.startStatus
              OR kran4Open.startStatus
              OR waitAfterKran4.startStatus
              OR kran5Close.startStatus
              OR didPKran1.startStatus
              OR kran1Open.startStatus
              OR kran2Open.startStatus
              OR kran3bClose.startStatus
              OR kran4Close.startStatus
              OR RunProtection_kr1.startStatus
              OR RunProtection_kr2.startStatus
              OR waitAfterKran5.startStatus
              OR testUnsuccessfulFilling.startStatus;

  StrAlg.Error:= BreakPuskTimer.errorStatus
              OR kran3bOpen.errorStatus
              OR kran4Open.errorStatus
              OR waitAfterKran4.errorStatus
              OR kran5Close.errorStatus
              OR didPKran1.errorStatus
              OR kran1Open.errorStatus
              OR kran2Open.errorStatus
              OR kran3bClose.errorStatus
              OR kran4Close.errorStatus
              OR RunProtection_kr1.errorStatus
              OR RunProtection_kr2.errorStatus
              OR waitAfterKran5.errorStatus
              OR testUnsuccessfulFilling.errorStatus;

  StrAlg.Top:=   BreakPuskTimer.topStatus
              OR kran3bOpen.topStatus
              OR kran4Open.topStatus
              OR waitAfterKran4.topStatus
              OR kran5Close.topStatus
              OR didPKran1.topStatus
              OR kran1Open.topStatus
              OR kran2Open.topStatus
              OR kran3bClose.topStatus
              OR kran4Close.topStatus
              OR RunProtection_kr1.topStatus
              OR RunProtection_kr2.topStatus
              OR waitAfterKran5.topStatus
              OR testUnsuccessfulFilling.topStatus;

  (*TODO: TYPE PROGRAM CODE HERE*)
  StrAlg.status :=  SHL(BYTE_TO_DWORD(source_for_Status), 29)
  			OR SHL(BYTE_TO_DWORD(cmd_for_Status), 26)
  			OR SHL(BYTE_TO_DWORD(command_error_for_Status), 23)
  			OR SHL(BOOL_TO_DWORD(StrAlg.OpcCommandsDisabled ), 21)
  			OR SHL(BOOL_TO_DWORD(StrAlg.hasError),4)
  			OR SHL(BOOL_TO_DWORD(StrAlg.CanRun),2)
  			OR SHL(BOOL_TO_DWORD(StrAlg.isEnded),1)
  			OR BOOL_TO_DWORD(StrAlg.isRuning);
END_FUNCTION_BLOCK

FUNCTION_BLOCK engineRunAlg
  VAR_IN_OUT
    StrAlg : struct_Alg;
  END_VAR
  VAR
    BreakPuskTimer : struct_PhaseAlgoritm;
    RunProtection_mvoff : struct_PhaseAlgoritm;
    LowOil_upStopust : struct_PhaseAlgoritm;
    mvOn : struct_PhaseAlgoritm;
    AutoPns_ph : struct_PhaseAlgoritm;
    AutoAvom_ph : struct_PhaseAlgoritm;
    pnsOff : struct_PhaseAlgoritm;
    testUnsuccessful : struct_PhaseAlgoritm;
    fb_BreakPuskTimer : fb_ph_Timer;
    fb_RunProtection_mvoff : fb_ph_DIprotection;
    fb_LowOil_upStopust : fb_ph_WaitAnalogValue;
    fb_mvOn : fb_ph_SectionSwitch;
    fb_AutoPns_ph : fb_ph_algoritm;
    fb_AutoAvom_ph : fb_ph_algoritm;
    fb_pnsOff : fb_ph_Switch;
    fb_testUnsuccessful : fb_ph_CustomPhase;
    _sunpackerCommand : fb_sunpackerCommand;
    _DualStateImAction : TYPE_DualStateImAction;
    _PhaseAlgoritmAction : TYPE_PhaseAlgoritmAction;
    source : BYTE;
    cmd : BYTE;
    lastCmd : BYTE;
    source_for_Status : BYTE;
    cmd_for_Status : BYTE;
    command_error_for_Status : BYTE;
    resetCmdTimer : TON;
    resetCmdTimerPriznak : BOOL;
    onInit : BOOL;
    waitReset : TON;
  END_VAR
  VAR_EXTERNAL
    IM : ImConfig;
    algoritms : AlgoritmsConfig;
    ai : AiConfig;
    protections : ProtectionsConfig;
    AlgTimers : struct_AlgTimers;
  END_VAR

  IF NOT onInit THEN

       fb_BreakPuskTimer(phaseNumber:=0, delay:=T#665S);
     fb_LowOil_upStopust(phaseNumber:=1);
                 fb_mvOn(phaseNumber:=2, act:=_on);
           fb_AutoPns_ph(phaseNumber:=3, act:=_run, waitCompletion:=FALSE);
          fb_AutoAvom_ph(phaseNumber:=4, act:=_run, waitCompletion:=FALSE);
               fb_pnsOff(phaseNumber:=5, act:=_off);
  fb_RunProtection_mvoff(phaseNumber:=7, act:=_run);
     fb_testUnsuccessful(phaseNumber:=17);

  onInit:=TRUE;
  END_IF;

          fb_BreakPuskTimer(StrPh:=BreakPuskTimer, timer:=AlgTimers.engineRun_BreakPuskTimer);
        fb_LowOil_upStopust(StrPh:=LowOil_upStopust, ai:=ai.P_masla_smazki_nizkoe, more:=im.AutoPns_UstStop.Value);
                    fb_mvOn(StrPh:=mvOn, Im:=Im.mv);
              fb_AutoPns_ph(StrPh:=AutoPns_ph, alg:=algoritms.AutoPns);
             fb_AutoAvom_ph(StrPh:=AutoAvom_ph, alg:=algoritms.AutoAvom);
                  fb_pnsOff(StrPh:=pnsOff, Im:=Im.pns);
     fb_RunProtection_mvoff(StrPh:=RunProtection_mvoff, StrDiP:=protections.mvOff);
        fb_testUnsuccessful(StrPh:=testUnsuccessful);

  StrAlg.CanRun := StrAlg.inCanRun;
  StrAlg.OpcCommandsDisabled := StrAlg.inOpcCommandsDisabled;

  IF StrAlg.isRuning THEN

      StrAlg.hasError := mvOn.error OR pnsOff.error OR testUnsuccessful.error;

      IF mvOn.top THEN
          runPhase(RunProtection_mvoff);
          runPhase(AutoAvom_ph);
          runPhase(LowOil_upStopust);
      END_IF;
      (*
      IF AutoAvom_ph.top THEN
          algoritms.AutoAvom.inOpcCommandsDisabled:=FALSE;
      END_IF;
      *)
      IF LowOil_upStopust.top THEN
          runPhase(pnsOff);
      END_IF;

      IF pnsOff.top THEN
         runPhase(AutoPns_ph);
      END_IF;

      IF BreakPuskTimer.top AND NOT AutoPns_ph.top THEN
            testUnsuccessful.error:=TRUE;
      END_IF;

      IF AutoPns_ph.top THEN
            resetPhase(BreakPuskTimer);
  	waitReset(IN:=TRUE, PT:= T#2S);
      END_IF;

      IF waitReset.Q AND NOT (algoritms.Apusk.isRuning OR algoritms.SemiAutoPusk.isRuning) THEN
  	resetIfRunning(StrAlg);
      END_IF;

      StrAlg.isEnded:= AutoPns_ph.top;
  END_IF;

  StrAlg.CanRun := StrAlg.inCanRun;
  StrAlg.OpcCommandsDisabled := StrAlg.inOpcCommandsDisabled;

  (* ---- Если управление с ВУ заблокировано, то  передаем команду из алгоритма ---- *)
  IF StrAlg.inOpcCommandsDisabled THEN
  	StrAlg.inCommand := StrAlg.inCommand_Alg;
  ELSE (* иначе передаем команду с АРМа*)
  	StrAlg.inCommand := StrAlg.inCommand_ARM;
  END_IF;

  _sunpackerCommand(command := StrAlg.inCommand);
  	source := _sunpackerCommand.source;
  	cmd := _sunpackerCommand.cmd;

  IF cmd <> 0 AND lastCmd <> cmd AND (((NOT StrAlg.opcCommandsDisabled) AND source > 0) OR source = 0) then
  	CASE BYTE_TO_INT(cmd) OF
  		(*cmdRun*) 1: 	IF (StrAlg.CanRun) THEN
  					StrAlg.isRuning := TRUE;
  					StrAlg.isEnded := FALSE;
  					StrAlg.hasError := FALSE;
  					(*****************       OnRun       *****************)

                                                    runPhase(mvOn);
                                                    runPhase(BreakPuskTimer);
                                                    runPhase(testUnsuccessful);

  					cmd_for_Status := cmd;
  					source_for_Status := source;
  					command_error_for_Status := 0;
  				ELSE
  					StrAlg.isRuning := FALSE;
  					StrAlg.isEnded := FALSE;
  					StrAlg.hasError 	:= FALSE;

  					cmd_for_Status := 0;
  					source_for_Status := source;
  					command_error_for_Status := cmd;
  				END_IF;
  		(*cmdReset*) 2: 	StrAlg.isRuning := FALSE;
  				StrAlg.isEnded := FALSE;
  				StrAlg.hasError 	:= FALSE;

                                           (*****************       OnReset       *****************)
                                          StrAlg.inCanRun:=FALSE;
                                          waitReset(IN:=FALSE);

                                          resetPhase(BreakPuskTimer);
                                          resetPhase(RunProtection_mvoff);
                                          resetPhase(LowOil_upStopust);
                                          resetPhase(mvOn);
                                          resetPhase(AutoPns_ph);
                                          resetPhase(AutoAvom_ph);
                                          resetPhase(pnsOff);
                                          resetPhase(testUnsuccessful);

  				cmd_for_Status := cmd;
  				source_for_Status := source;
  				command_error_for_Status := 0;
  	END_CASE;
  	resetCmdTimer(IN := false);
  	resetCmdTimerPriznak := TRUE;
  END_IF;
  lastCmd := cmd;

  resetCmdTimer(IN := resetCmdTimerPriznak, PT := T#5S);
  IF resetCmdTimer.Q THEN
  	resetCmdTimerPriznak := FALSE;
  	source_for_Status := 0;
  	cmd_for_Status := 0;
  	command_error_for_Status := 0;
  END_IF;

  StrAlg.Start:= BreakPuskTimer.startStatus
              OR RunProtection_mvoff.startStatus
              OR LowOil_upStopust.startStatus
              OR mvOn.startStatus
              OR AutoPns_ph.startStatus
              OR AutoAvom_ph.startStatus
              OR pnsOff.startStatus
              OR testUnsuccessful.startStatus;

  StrAlg.Error:= BreakPuskTimer.errorStatus
              OR RunProtection_mvoff.errorStatus
              OR LowOil_upStopust.errorStatus
              OR mvOn.errorStatus
              OR AutoPns_ph.errorStatus
              OR AutoAvom_ph.errorStatus
              OR pnsOff.errorStatus
              OR testUnsuccessful.errorStatus;

  StrAlg.Top:=   BreakPuskTimer.topStatus
              OR RunProtection_mvoff.topStatus
              OR LowOil_upStopust.topStatus
              OR mvOn.topStatus
              OR AutoPns_ph.topStatus
              OR AutoAvom_ph.topStatus
              OR pnsOff.topStatus
              OR testUnsuccessful.topStatus;

  (*TODO: TYPE PROGRAM CODE HERE*)
  StrAlg.status :=  SHL(BYTE_TO_DWORD(source_for_Status), 29)
  			OR SHL(BYTE_TO_DWORD(cmd_for_Status), 26)
  			OR SHL(BYTE_TO_DWORD(command_error_for_Status), 23)
  			OR SHL(BOOL_TO_DWORD(StrAlg.OpcCommandsDisabled ), 21)
  			OR SHL(BOOL_TO_DWORD(StrAlg.hasError),4)
  			OR SHL(BOOL_TO_DWORD(StrAlg.CanRun),2)
  			OR SHL(BOOL_TO_DWORD(StrAlg.isEnded),1)
  			OR BOOL_TO_DWORD(StrAlg.isRuning);
END_FUNCTION_BLOCK

FUNCTION_BLOCK puskKalg
  VAR_IN_OUT
    StrAlg : struct_Alg;
  END_VAR
  VAR
    puskOilSystem : struct_PhaseAlgoritm;
  END_VAR
  VAR_IN_OUT
    questionFilling : struct_Question;
  END_VAR
  VAR
    filling : struct_PhaseAlgoritm;
  END_VAR
  VAR_IN_OUT
    questionUnload : struct_Question;
  END_VAR
  VAR
    kran3bOpen : struct_PhaseAlgoritm;
    kran4Close : struct_PhaseAlgoritm;
    kran1Close : struct_PhaseAlgoritm;
    kran2Close : struct_PhaseAlgoritm;
    kran5open : struct_PhaseAlgoritm;
    wait720 : struct_PhaseAlgoritm;
    noGasInPipe : struct_PhaseAlgoritm;
    AutoNUoff : struct_PhaseAlgoritm;
    nu1Off : struct_PhaseAlgoritm;
    nu2Off : struct_PhaseAlgoritm;
    pnsWaitOff : struct_PhaseAlgoritm;
    testUnsuccessfulUnfill : struct_PhaseAlgoritm;
    fb_puskOilSystem : fb_ph_algoritm;
    fb_questionFilling : fb_Question;
    fb_filling : fb_ph_algoritm;
    fb_questionUnload : fb_Question;
    fb_kran3bOpen : fb_ph_Kran;
    fb_kran4Close : fb_ph_CustomPhase;
    fb_kran1Close : fb_ph_Kran;
    fb_kran2Close : fb_ph_Kran;
    fb_kran5open : fb_ph_Kran;
    fb_wait720 : fb_ph_Timer;
    fb_noGasInPipe : fb_ph_CustomPhase;
    fb_AutoNUoff : fb_ph_algoritm;
    fb_nu1Off : fb_ph_OilPump;
    fb_nu2Off : fb_ph_OilPump;
    fb_pnsWaitOff : fb_ph_algoritm;
    fb_testUnsuccessfulUnfill : fb_ph_CustomPhase;
    _sunpackerCommand : fb_sunpackerCommand;
    _DualStateImAction : TYPE_DualStateImAction;
    _Answers : TYPE_Answers;
    _statusDualInput : TYPE_statusDualInput;
    _StatusAi : TYPE_StatusAi;
    _PhaseAlgoritmAction : TYPE_PhaseAlgoritmAction;
    source : BYTE;
    cmd : BYTE;
    lastCmd : BYTE;
    source_for_Status : BYTE;
    cmd_for_Status : BYTE;
    command_error_for_Status : BYTE;
    resetCmdTimer : TON;
    resetCmdTimerPriznak : BOOL;
  END_VAR
  VAR CONSTANT
    Ust_Pgaza : LREAL := 0.3;
  END_VAR
  VAR
    OpcCommandsKransEnabled : BOOL;
    OpcCommandsKransDisabled : BOOL;
    _resetQuestion1 : BOOL;
    _resetQuestion2 : BOOL;
    onInit : BOOL;
    waitReset : TON;
  END_VAR
  VAR_EXTERNAL
    IM : ImConfig;
    algoritms : AlgoritmsConfig;
    ai : AiConfig;
    AlgTimers : struct_AlgTimers;
    ModeGpa : TYPE_ModeGpa;
    algManager : struct_AlgoritmsManager;
    protections : ProtectionsConfig;
  END_VAR

  IF NOT onInit THEN

            fb_puskOilSystem(phaseNumber:=0, act:=_run, waitCompletion:=TRUE);
        questionFilling.AnswerVariants:=_Answers.ANS_YES;
                  fb_filling(phaseNumber:=1, act:=_run, waitCompletion:=TRUE);
      questionUnload.AnswerVariants:=_Answers.ANS_YES;
               fb_kran3bOpen(phaseNumber:=3, act:=_on);
               fb_kran4Close(phaseNumber:=4);
               fb_kran1Close(phaseNumber:=5, act:=_off);
               fb_kran2Close(phaseNumber:=6, act:=_off);
                fb_kran5open(phaseNumber:=7, act:=_on);
                  fb_wait720(phaseNumber:=8, delay:=T#720S);
              fb_noGasInPipe(phaseNumber:=9);
                fb_AutoNUoff(phaseNumber:=10, act:=_reset, waitCompletion:=FALSE);
                   fb_nu1Off(phaseNumber:=11, act:=_off);
                   fb_nu2Off(phaseNumber:=12, act:=_off);
               fb_pnsWaitOff(phaseNumber:=15, act:=_run, waitCompletion:=TRUE);
   fb_testUnsuccessfulUnfill(phaseNumber:=18);

  onInit:=TRUE;
  END_IF;

            fb_puskOilSystem(StrPh:=puskOilSystem, alg:=algoritms.puskOilSystem);
          fb_questionFilling(StrQ:=questionFilling);
                  fb_filling(StrPh:=filling, alg:=algoritms.filling);
           fb_questionUnload(StrQ:=questionUnload);
               fb_kran3bOpen(StrPh:=kran3bOpen, Im:=Im.kran3b);
               fb_kran4Close(StrPh:=kran4Close);
               fb_kran1Close(StrPh:=kran1Close, Im:=Im.kran1);
               fb_kran2Close(StrPh:=kran2Close, Im:=Im.kran2);
                fb_kran5open(StrPh:=kran5open, Im:=Im.kran5);
                  fb_wait720(StrPh:=wait720, timer:=AlgTimers.puskK_wait720);
              fb_noGasInPipe(StrPh:=noGasInPipe);
                fb_AutoNUoff(StrPh:=AutoNUoff, alg:=algoritms.autoNu);
                   fb_nu1Off(StrPh:=nu1Off, Im:=Im.nu1);
                   fb_nu2Off(StrPh:=nu2Off, Im:=Im.nu2);
               fb_pnsWaitOff(StrPh:=pnsWaitOff, alg:=algoritms.vibegPNS);
   fb_testUnsuccessfulUnfill(StrPh:=testUnsuccessfulUnfill);

  StrAlg.CanRun := StrAlg.inCanRun;
  StrAlg.OpcCommandsDisabled := StrAlg.inOpcCommandsDisabled;

  IF StrAlg.isRuning THEN

      StrAlg.hasError := kran3bOpen.error OR kran1Close.error OR kran2Close.error OR kran5open.error OR testUnsuccessfulUnfill.error;

      IF puskOilSystem.top THEN
           IF NOT _resetQuestion1 THEN
           askQuestion(questionFilling);
           _resetQuestion1:=TRUE;
           END_IF;
      END_IF;

      IF questionFilling.answer = _Answers.ANS_YES THEN
          runPhase(filling);
          resetQuestion(questionFilling);
      END_IF;

      IF filling.top THEN
         OpcCommandsKransEnabled:=TRUE;
         resetDiProtection(protections.Kran1sdvig);
         resetDiProtection(protections.Kran2sdvig);
         IF NOT _resetQuestion2 THEN
         askQuestion(questionUnload);
         _resetQuestion2:=TRUE;
         END_IF;
      END_IF;

       IF questionUnload.answer = _Answers.ANS_YES THEN
          OpcCommandsKransDisabled:=TRUE;
          runPhase(kran3bOpen);
          runPhase(wait720);
          resetQuestion(questionUnload);
      END_IF;

      IF kran3bOpen.top THEN
            resetDiProtection(protections.Kran1sdvig);
            resetDiProtection(protections.Kran2sdvig);

            runPhase(kran1Close);
            runPhase(kran2Close);
            runPhase(kran4Close);
      END_IF;

       IF kran4Close.start AND NOT kran4Close.top THEN
  	kran4Close.top:= Im.kran4.onStatus = _statusDualInput.STATUS_OFF;
      END_IF;

      IF kran1Close.top AND kran2Close.top AND kran4Close.top THEN
  	runPhase(kran5open);
      END_IF;

      IF kran5open.top THEN
  	runPhase(noGasInPipe);
      END_IF;

      IF noGasInPipe.start AND (NOT noGasInPipe.top) THEN
  	noGasInPipe.top:=  (ai.P_gaza_na_vkhode_nagnetatelia.interval >= _statusAi.NORMAL
                           AND  ai.P_gaza_na_vkhode_nagnetatelia.value< Ust_Pgaza )
                           AND (ai.P_gaza_na_vykhode_nagnetatelia.interval >= _statusAi.NORMAL
                           AND  ai.P_gaza_na_vykhode_nagnetatelia.value< Ust_Pgaza);
      END_IF;

      IF noGasInPipe.top THEN

            ai.dPmaslo_gaz.Disabled_LA:=TRUE;
            ai.dPmaslo_gaz.Disabled_LW:=TRUE;
            IM.SingleSignals.dP_oilgaz_low.Disabled_Sig:=TRUE;
            resetAiProtection(protections.dP_maslogaz_LA);
            resetDiProtection(protections.dP_masloGaz_LowDI);
  	runPhase(AutoNUoff);

      END_IF;

       IF autoNuOff.top THEN
  	runPhase(nu1off);
            runPhase(nu2off);
      END_IF;

      IF nu1Off.top AND nu2Off.top THEN
  	runPhase(pnsWaitOff);
      END_IF;

      IF wait720.top AND NOT (pnsWaitOff.top) THEN
            testUnsuccessfulUnfill.error:=TRUE;
      END_IF;

      IF pnsWaitOff.top THEN
            resetPhase(wait720);
  	waitReset(IN:=TRUE, PT:= T#3S);
      END_IF;

      IF waitReset.Q THEN
          resetIfRunning(algoritms.vibegPNS);
          algManager.nMode:=ModeGpa.MODE_STOP;
          resetIfRunning(StrAlg);
      END_IF;

      StrAlg.isEnded:= pnsWaitOff.top;

      IF OpcCommandsKransEnabled AND NOT OpcCommandsKransDisabled THEN
  	IF      (im.pns.onStatus = _statusDualInput.STATUS_ON)
                AND (im.nu1.onStatus = _statusDualInput.STATUS_ON OR im.nu2.onStatus = _statusDualInput.STATUS_ON)
  	    AND (ai.dPmaslo_gaz.interval >= _statusAi.normal)
                AND (ai.dPmaslo_gaz.value > im.PuskOilSystem_UstdPmg.Value)
            THEN
  	    IM.Kran3b.inOpcCommandsDisabled:=FALSE;
  	    Im.kran4.inOpcCommandsDisabled:=FALSE;
  	    Im.kran5.inOpcCommandsDisabled:=FALSE;
  		IF	Im.SingleSignals.dP_gazgaz_Kran1.q THEN
  			Im.kran1.inOpcCommandsDisabled:=FALSE;
  			Im.kran2.inOpcCommandsDisabled:=FALSE;
  		ELSE
  			Im.kran1.inOpcCommandsDisabled:=TRUE;
  			Im.kran2.inOpcCommandsDisabled:=TRUE;
  		END_IF;
            ELSE
  	    Im.kran1.inOpcCommandsDisabled:=TRUE;
  	    Im.kran2.inOpcCommandsDisabled:=TRUE;
  	    Im.kran3b.inOpcCommandsDisabled:=TRUE;
  	    Im.kran4.inOpcCommandsDisabled:=TRUE;
  	    Im.kran5.inOpcCommandsDisabled:=TRUE;
            END_IF;

      ELSE
  	Im.kran1.inOpcCommandsDisabled:=TRUE;
  	Im.kran2.inOpcCommandsDisabled:=TRUE;
  	Im.kran3b.inOpcCommandsDisabled:=TRUE;
  	Im.kran4.inOpcCommandsDisabled:=TRUE;
  	Im.kran5.inOpcCommandsDisabled:=TRUE;
      END_IF;
  END_IF;

  StrAlg.CanRun := StrAlg.inCanRun;
  StrAlg.OpcCommandsDisabled := StrAlg.inOpcCommandsDisabled;

  (* ---- Если управление с ВУ заблокировано, то  передаем команду из алгоритма ---- *)
  IF StrAlg.inOpcCommandsDisabled THEN
  	StrAlg.inCommand := StrAlg.inCommand_Alg;
  ELSE (* иначе передаем команду с АРМа*)
  	StrAlg.inCommand := StrAlg.inCommand_ARM;
  END_IF;

  _sunpackerCommand(command := StrAlg.inCommand);
  	source := _sunpackerCommand.source;
  	cmd := _sunpackerCommand.cmd;

  IF cmd <> 0 AND lastCmd <> cmd AND (((NOT StrAlg.opcCommandsDisabled) AND source > 0) OR source = 0) then
  	CASE BYTE_TO_INT(cmd) OF
  		(*cmdRun*) 1: 	IF (StrAlg.CanRun) THEN
  					StrAlg.isRuning := TRUE;
  					StrAlg.isEnded := FALSE;
  					StrAlg.hasError := FALSE;
  					(*****************       OnRun       *****************)

                                                    algManager.nMode:=ModeGpa.MODE_PUSKK;
                                                    resetAndDisable(alg:=algoritms.ppu);
                                                    algoritms.puskOilSystem.inCanRun:= TRUE;
                                                    algoritms.filling.inCanRun:= TRUE;
                                                    runPhase(puskOilSystem);

  					cmd_for_Status := cmd;
  					source_for_Status := source;
  					command_error_for_Status := 0;
  				ELSE
  					StrAlg.isRuning := FALSE;
  					StrAlg.isEnded := FALSE;
  					StrAlg.hasError 	:= FALSE;

  					cmd_for_Status := 0;
  					source_for_Status := source;
  					command_error_for_Status := cmd;
  				END_IF;
  		(*cmdReset*) 2: 	StrAlg.isRuning := FALSE;
  				StrAlg.isEnded := FALSE;
  				StrAlg.hasError 	:= FALSE;

                                           (*****************       OnReset       *****************)
                                          OpcCommandsKransEnabled:=FALSE;
                                          OpcCommandsKransDisabled:=FALSE;
                                          waitReset(IN:=FALSE);
                                          _resetQuestion1:=FALSE;
                                          _resetQuestion2:=FALSE;
                                          resetPhase(puskOilSystem);
                                          resetPhase(filling);
                                          resetPhase(kran3bOpen);
                                          resetPhase(kran4Close);
                                          resetPhase(kran1Close);
                                          resetPhase(kran2Close);
                                          resetPhase(kran5open);
                                          resetPhase(wait720);
                                          resetPhase(noGasInPipe);
                                          resetPhase(AutoNUoff);
                                          resetPhase(nu1Off);
                                          resetPhase(nu2Off);
                                          resetPhase(pnsWaitOff);
                                          resetPhase(testUnsuccessfulUnfill);
                                          BlockAllIM(IM);
                                          resetQuestion(questionFilling);
                                          resetQuestion(questionUnload);

                                          StrAlg.inOpcCommandsDisabled:=FALSE;

  				cmd_for_Status := cmd;
  				source_for_Status := source;
  				command_error_for_Status := 0;
  	END_CASE;
  	resetCmdTimer(IN := false);
  	resetCmdTimerPriznak := TRUE;
  END_IF;
  lastCmd := cmd;

  resetCmdTimer(IN := resetCmdTimerPriznak, PT := T#5S);
  IF resetCmdTimer.Q THEN
  	resetCmdTimerPriznak := FALSE;
  	source_for_Status := 0;
  	cmd_for_Status := 0;
  	command_error_for_Status := 0;
  END_IF;

  StrAlg.Start:= puskOilSystem.startStatus
              OR filling.startStatus
              OR kran3bOpen.startStatus
              OR kran4Close.startStatus
              OR kran1Close.startStatus
              OR kran2Close.startStatus
              OR kran5open.startStatus
              OR wait720.startStatus
              OR noGasInPipe.startStatus
              OR AutoNUoff.startStatus
              OR nu1Off.startStatus
              OR nu2Off.startStatus
              OR pnsWaitOff.startStatus
              OR testUnsuccessfulUnfill.startStatus;

  StrAlg.Error:=  puskOilSystem.errorStatus
              OR filling.errorStatus
              OR kran3bOpen.errorStatus
              OR kran4Close.errorStatus
              OR kran1Close.errorStatus
              OR kran2Close.errorStatus
              OR kran5open.errorStatus
              OR wait720.errorStatus
              OR noGasInPipe.errorStatus
              OR AutoNUoff.errorStatus
              OR nu1Off.errorStatus
              OR nu2Off.errorStatus
              OR pnsWaitOff.errorStatus
              OR testUnsuccessfulUnfill.errorStatus;

  StrAlg.Top:=   puskOilSystem.topStatus
              OR filling.topStatus
              OR kran3bOpen.topStatus
              OR kran4Close.topStatus
              OR kran1Close.topStatus
              OR kran2Close.topStatus
              OR kran5open.topStatus
              OR wait720.topStatus
              OR noGasInPipe.topStatus
              OR AutoNUoff.topStatus
              OR nu1Off.topStatus
              OR nu2Off.topStatus
              OR pnsWaitOff.topStatus
              OR testUnsuccessfulUnfill.topStatus;

  (*TODO: TYPE PROGRAM CODE HERE*)
  StrAlg.status :=  SHL(BYTE_TO_DWORD(source_for_Status), 29)
  			OR SHL(BYTE_TO_DWORD(cmd_for_Status), 26)
  			OR SHL(BYTE_TO_DWORD(command_error_for_Status), 23)
  			OR SHL(BOOL_TO_DWORD(StrAlg.OpcCommandsDisabled ), 21)
  			OR SHL(BOOL_TO_DWORD(StrAlg.hasError),4)
  			OR SHL(BOOL_TO_DWORD(StrAlg.CanRun),2)
  			OR SHL(BOOL_TO_DWORD(StrAlg.isEnded),1)
  			OR BOOL_TO_DWORD(StrAlg.isRuning);
END_FUNCTION_BLOCK

FUNCTION_BLOCK puskValg
  VAR_IN_OUT
    StrAlg : struct_Alg;
  END_VAR
  VAR
    puskOilSystem : struct_PhaseAlgoritm;
  END_VAR
  VAR_IN_OUT
    questionEngine : struct_Question;
  END_VAR
  VAR
    runningEngine : struct_PhaseAlgoritm;
  END_VAR
  VAR_IN_OUT
    questionMVoff : struct_Question;
  END_VAR
  VAR
    mvOff : struct_PhaseAlgoritm;
    pnsOn : struct_PhaseAlgoritm;
    wait600 : struct_PhaseAlgoritm;
    AutoNUoff : struct_PhaseAlgoritm;
    nu1Off : struct_PhaseAlgoritm;
    nu2Off : struct_PhaseAlgoritm;
    autoAvomOff : struct_PhaseAlgoritm;
    Avom1Off : struct_PhaseAlgoritm;
    Avom2Off : struct_PhaseAlgoritm;
    pnsWaitOff : struct_PhaseAlgoritm;
    testUnsuccessful : struct_PhaseAlgoritm;
    fb_puskOilSystem : fb_ph_algoritm;
    fb_questionEngine : fb_Question;
    fb_runningEngine : fb_ph_algoritm;
    fb_questionMVoff : fb_Question;
    fb_mvOff : fb_ph_SectionSwitch;
    fb_pnsOn : fb_ph_Switch;
    fb_wait600 : fb_ph_Timer;
    fb_AutoNUoff : fb_ph_algoritm;
    fb_nu1Off : fb_ph_OilPump;
    fb_nu2Off : fb_ph_OilPump;
    fb_autoAvomOff : fb_ph_algoritm;
    fb_Avom1Off : fb_ph_Switch;
    fb_Avom2Off : fb_ph_Switch;
    fb_pnsWaitOff : fb_ph_algoritm;
    fb_testUnsuccessful : fb_ph_CustomPhase;
    _sunpackerCommand : fb_sunpackerCommand;
    _DualStateImAction : TYPE_DualStateImAction;
    _Answers : TYPE_Answers;
    _statusDualInput : TYPE_statusDualInput;
    _StatusAi : TYPE_StatusAi;
    _PhaseAlgoritmAction : TYPE_PhaseAlgoritmAction;
    source : BYTE;
    cmd : BYTE;
    lastCmd : BYTE;
    source_for_Status : BYTE;
    cmd_for_Status : BYTE;
    command_error_for_Status : BYTE;
    resetCmdTimer : TON;
    resetCmdTimerPriznak : BOOL;
  END_VAR
  VAR CONSTANT
    Ust_Pgaza : LREAL := 0.3;
  END_VAR
  VAR
    onInit : BOOL;
    _resetQuestion1 : BOOL;
    _resetQuestion2 : BOOL;
    waitReset : TON;
  END_VAR
  VAR_EXTERNAL
    IM : ImConfig;
    algoritms : AlgoritmsConfig;
    ai : AiConfig;
    AlgTimers : struct_AlgTimers;
    ModeGpa : TYPE_ModeGpa;
    algManager : struct_AlgoritmsManager;
    protections : ProtectionsConfig;
  END_VAR

  IF NOT onInit THEN

            fb_puskOilSystem(phaseNumber:=0, act:=_run, waitCompletion:=TRUE);
         questionEngine.AnswerVariants:=_Answers.ANS_YES;
            fb_runningEngine(phaseNumber:=1, act:=_run, waitCompletion:=TRUE);
          questionMVoff.AnswerVariants:=_Answers.ANS_YES;
                    fb_mvOff(phaseNumber:=3, act:=_off);
                    fb_pnsOn(phaseNumber:=4, act:=_on);
                  fb_wait600(phaseNumber:=8, delay:=T#600S);
                fb_AutoNUoff(phaseNumber:=10, act:=_reset, waitCompletion:=FALSE);
                   fb_nu1Off(phaseNumber:=11, act:=_off);
                   fb_nu2Off(phaseNumber:=12, act:=_off);
               fb_pnsWaitOff(phaseNumber:=15, act:=_run, waitCompletion:=TRUE);
              fb_autoAvomOff(phaseNumber:=7, act:=_reset, waitCompletion:=FALSE);
                 fb_Avom1Off(phaseNumber:=5, act:=_off);
                 fb_Avom2Off(phaseNumber:=6, act:=_off);
         fb_testUnsuccessful(phaseNumber:=17);

  onInit:=TRUE;
  END_IF;

            fb_puskOilSystem(StrPh:=puskOilSystem, alg:=algoritms.puskOilSystem);
           fb_questionEngine(StrQ:=questionEngine);
            fb_runningEngine(StrPh:=runningEngine, alg:=algoritms.engineRun);
            fb_questionMVoff(StrQ:=questionMVoff);
                    fb_mvOff(StrPh:=mvOff, Im:=Im.mv);
                    fb_pnsOn(StrPh:=pnsOn, Im:=Im.pns);
                  fb_wait600(StrPh:=wait600, timer:=AlgTimers.puskV_wait600);
                fb_AutoNUoff(StrPh:=AutoNUoff, alg:=algoritms.autoNu);
                   fb_nu1Off(StrPh:=nu1Off, Im:=Im.nu1);
                   fb_nu2Off(StrPh:=nu2Off, Im:=Im.nu2);
               fb_pnsWaitOff(StrPh:=pnsWaitOff, alg:=algoritms.vibegPNS);
              fb_autoAvomOff(StrPh:=autoAvomOff, alg:=algoritms.AutoAvom);
                 fb_Avom1Off(StrPh:=Avom1Off, Im:=Im.v1_Avom);
                 fb_Avom2Off(StrPh:=Avom2Off, Im:=Im.v2_Avom);
         fb_testUnsuccessful(StrPh:=testUnsuccessful);

  StrAlg.CanRun := StrAlg.inCanRun;
  StrAlg.OpcCommandsDisabled := StrAlg.inOpcCommandsDisabled;

  IF StrAlg.isRuning THEN

      StrAlg.hasError := mvOff.error OR pnsOn.error OR testUnsuccessful.error;

      IF puskOilSystem.top THEN
           IF NOT _resetQuestion1 THEN
           askQuestion(questionEngine);
           _resetQuestion1:=TRUE;
           END_IF;
      END_IF;

      IF questionEngine.answer = _Answers.ANS_YES THEN
          runPhase(runningEngine);
          resetQuestion(questionEngine);
      END_IF;

      IF runningEngine.top THEN
         IF NOT _resetQuestion2 THEN
         askQuestion(questionMVoff);
         _resetQuestion2:=TRUE;
         END_IF;
      END_IF;

       IF questionMVoff.answer = _Answers.ANS_YES THEN

          resetDiProtection(protections.mvOff);
          resetIfRunning(algoritms.AutoPns);
          runPhase(mvOff);
          runPhase(wait600);
          resetQuestion(questionMVoff);
       END_IF;

      IF mvOff.top THEN
          runPhase(pnsOn);
      END_IF;

      IF pnsOn.top THEN

            ai.dPmaslo_gaz.Disabled_LA:=TRUE;
            ai.dPmaslo_gaz.Disabled_LW:=TRUE;
            IM.SingleSignals.dP_oilgaz_low.Disabled_Sig:=TRUE;
            resetAiProtection(protections.dP_maslogaz_LA);
            resetDiProtection(protections.dP_masloGaz_LowDI);
  	runPhase(AutoNUoff);

      END_IF;

       IF autoNuOff.top THEN
  	runPhase(nu1off);
            runPhase(nu2off);
      END_IF;

      IF nu1Off.top AND nu2Off.top THEN
  	runPhase(pnsWaitOff);
      END_IF;

      IF wait600.top AND NOT (pnsWaitOff.top) THEN
            testUnsuccessful.error:=TRUE;
      END_IF;

      IF pnsWaitOff.top THEN
            resetPhase(wait600);
            runPhase(autoAvomOff);
  	waitReset(IN:=TRUE, PT:= T#3S);
      END_IF;

      IF autoAvomOff.top THEN
            runPhase(Avom1Off);
            runPhase(Avom2Off);
      END_IF;

      IF waitReset.Q THEN
          resetIfRunning(algoritms.vibegPNS);
          algManager.nMode:=ModeGpa.MODE_STOP;
          resetIfRunning(StrAlg);
      END_IF;

      StrAlg.isEnded:= pnsWaitOff.top;

  END_IF;

  StrAlg.CanRun := StrAlg.inCanRun;
  StrAlg.OpcCommandsDisabled := StrAlg.inOpcCommandsDisabled;

  (* ---- Если управление с ВУ заблокировано, то  передаем команду из алгоритма ---- *)
  IF StrAlg.inOpcCommandsDisabled THEN
  	StrAlg.inCommand := StrAlg.inCommand_Alg;
  ELSE (* иначе передаем команду с АРМа*)
  	StrAlg.inCommand := StrAlg.inCommand_ARM;
  END_IF;

  _sunpackerCommand(command := StrAlg.inCommand);
  	source := _sunpackerCommand.source;
  	cmd := _sunpackerCommand.cmd;

  IF cmd <> 0 AND lastCmd <> cmd AND (((NOT StrAlg.opcCommandsDisabled) AND source > 0) OR source = 0) then
  	CASE BYTE_TO_INT(cmd) OF
  		(*cmdRun*) 1: 	IF (StrAlg.CanRun) THEN
  					StrAlg.isRuning := TRUE;
  					StrAlg.isEnded := FALSE;
  					StrAlg.hasError := FALSE;
  					(*****************       OnRun       *****************)

                                                    algManager.nMode:=ModeGpa.MODE_PUSKV;
                                                    resetAndDisable(alg:=algoritms.ppu);
                                                    algoritms.puskOilSystem.inCanRun:= TRUE;
                                                    algoritms.engineRun.inCanRun:= TRUE;
                                                    runPhase(puskOilSystem);

  					cmd_for_Status := cmd;
  					source_for_Status := source;
  					command_error_for_Status := 0;
  				ELSE
  					StrAlg.isRuning := FALSE;
  					StrAlg.isEnded := FALSE;
  					StrAlg.hasError 	:= FALSE;

  					cmd_for_Status := 0;
  					source_for_Status := source;
  					command_error_for_Status := cmd;
  				END_IF;
  		(*cmdReset*) 2: 	StrAlg.isRuning := FALSE;
  				StrAlg.isEnded := FALSE;
  				StrAlg.hasError 	:= FALSE;

                                           (*****************       OnReset       *****************)
                                          waitReset(IN:=FALSE);
                                          _resetQuestion1:=FALSE;
                                          _resetQuestion2:=FALSE;
                                          resetPhase(puskOilSystem);
                                          resetPhase(runningEngine);
                                          resetPhase(mvOff);
                                          resetPhase(pnsOn);
                                          resetPhase(wait600);
                                          resetPhase(AutoNUoff);
                                          resetPhase(nu1Off);
                                          resetPhase(nu2Off);
                                          resetPhase(pnsWaitOff);
  	                              resetPhase(autoAvomOff);
                                          resetPhase(Avom1Off);
                                          resetPhase(Avom2Off);
                                          resetPhase(testUnsuccessful);

                                          resetQuestion(questionEngine);
                                          resetQuestion(questionMVoff);

                                          StrAlg.inOpcCommandsDisabled:=FALSE;

  				cmd_for_Status := cmd;
  				source_for_Status := source;
  				command_error_for_Status := 0;
  	END_CASE;
  	resetCmdTimer(IN := false);
  	resetCmdTimerPriznak := TRUE;
  END_IF;
  lastCmd := cmd;

  resetCmdTimer(IN := resetCmdTimerPriznak, PT := T#5S);
  IF resetCmdTimer.Q THEN
  	resetCmdTimerPriznak := FALSE;
  	source_for_Status := 0;
  	cmd_for_Status := 0;
  	command_error_for_Status := 0;
  END_IF;

  StrAlg.Start:= puskOilSystem.startStatus
              OR runningEngine.startStatus
              OR mvOff.startStatus
              OR pnsOn.startStatus
              OR wait600.startStatus
              OR AutoNUoff.startStatus
              OR nu1Off.startStatus
              OR nu2Off.startStatus
              OR pnsWaitOff.startStatus
              OR testUnsuccessful.startStatus;

  StrAlg.Error:=  puskOilSystem.errorStatus
              OR runningEngine.errorStatus
              OR mvOff.errorStatus
              OR pnsOn.errorStatus
              OR wait600.errorStatus
              OR AutoNUoff.errorStatus
              OR nu1Off.errorStatus
              OR nu2Off.errorStatus
              OR pnsWaitOff.errorStatus
              OR testUnsuccessful.errorStatus;

  StrAlg.Top:=   puskOilSystem.topStatus
              OR runningEngine.topStatus
              OR mvOff.topStatus
              OR pnsOn.topStatus
              OR wait600.topStatus
              OR AutoNUoff.topStatus
              OR nu1Off.topStatus
              OR nu2Off.topStatus
              OR pnsWaitOff.topStatus
              OR testUnsuccessful.topStatus;

  (*TODO: TYPE PROGRAM CODE HERE*)
  StrAlg.status :=  SHL(BYTE_TO_DWORD(source_for_Status), 29)
  			OR SHL(BYTE_TO_DWORD(cmd_for_Status), 26)
  			OR SHL(BYTE_TO_DWORD(command_error_for_Status), 23)
  			OR SHL(BOOL_TO_DWORD(StrAlg.OpcCommandsDisabled ), 21)
  			OR SHL(BOOL_TO_DWORD(StrAlg.hasError),4)
  			OR SHL(BOOL_TO_DWORD(StrAlg.CanRun),2)
  			OR SHL(BOOL_TO_DWORD(StrAlg.isEnded),1)
  			OR BOOL_TO_DWORD(StrAlg.isRuning);
END_FUNCTION_BLOCK

FUNCTION_BLOCK testdPmgAlg
  VAR_IN_OUT
    StrAlg : struct_Alg;
  END_VAR
  VAR
    puskOilSystem : struct_PhaseAlgoritm;
  END_VAR
  VAR_IN_OUT
    algContinue : struct_Question;
  END_VAR
  VAR
    nuOff : struct_PhaseAlgoritm;
    dPmgAi : struct_PhaseAlgoritm;
    dPmgDi : struct_PhaseAlgoritm;
    nuOn : struct_PhaseAlgoritm;
    noRezrv : struct_PhaseAlgoritm;
    BreakTest : struct_PhaseAlgoritm;
    testUnsuccessful : struct_PhaseAlgoritm;
    pnsOff : struct_PhaseAlgoritm;
    stopANU : struct_PhaseAlgoritm;
    Ust_dPLow : struct_PhaseAlgoritm;
    nu1Off : struct_PhaseAlgoritm;
    nu2Off : struct_PhaseAlgoritm;
    stopNU1 : struct_PhaseAlgoritm;
    stopNU2 : struct_PhaseAlgoritm;
    fb_puskOilSystem : fb_ph_algoritm;
    fb_algContinue : fb_Question;
    fb_nuOff : fb_ph_CustomPhase;
    fb_dPmgAi : fb_ph_WaitAnalogValue;
    fb_dPmgDi : fb_ph_CustomPhase;
    fb_nuOn : fb_ph_CustomPhase;
    fb_noRezrv : fb_ph_CustomPhase;
    fb_BreakTest : fb_ph_Timer;
    fb_testUnsuccessful : fb_ph_CustomPhase;
    fb_pnsOff : fb_ph_Switch;
    fb_stopANU : fb_ph_CustomPhase;
    fb_nu1Off : fb_ph_OilPump;
    fb_nu2Off : fb_ph_OilPump;
    fb_stopNU1 : fb_ph_OilPump;
    fb_stopNU2 : fb_ph_OilPump;
    _sunpackerCommand : fb_sunpackerCommand;
    _DualStateImAction : TYPE_DualStateImAction;
    _Answers : TYPE_Answers;
    _statusDualInput : TYPE_statusDualInput;
    _StatusAi : TYPE_StatusAi;
    _PhaseAlgoritmAction : TYPE_PhaseAlgoritmAction;
    source : BYTE;
    cmd : BYTE;
    lastCmd : BYTE;
    source_for_Status : BYTE;
    cmd_for_Status : BYTE;
    command_error_for_Status : BYTE;
    resetCmdTimer : TON;
    resetCmdTimerPriznak : BOOL;
    onInit : BOOL;
    _resetQuestion : BOOL;
    waitReset : TON;
    WaitOnNU : TON;
  END_VAR
  VAR_EXTERNAL
    IM : ImConfig;
    algoritms : AlgoritmsConfig;
    ai : AiConfig;
    AlgTimers : struct_AlgTimers;
    ModeGpa : TYPE_ModeGpa;
    algManager : struct_AlgoritmsManager;
    protections : ProtectionsConfig;
    NotHasRezervNU : BOOL;
  END_VAR

  IF NOT onInit THEN

      fb_puskOilSystem(phaseNumber:=0, act:=_run, waitCompletion:=TRUE);
          algContinue.AnswerVariants:=_Answers.ANS_YES;
              fb_nuOff(phaseNumber:=1);
             fb_dPmgAi(phaseNumber:=2);
             fb_dPmgDi(phaseNumber:=3);
               fb_nuOn(phaseNumber:=4);
            fb_noRezrv(phaseNumber:=5);
   fb_testUnsuccessful(phaseNumber:=6);
          fb_BreakTest(phaseNumber:=7, delay:=T#10S);
             fb_pnsOff(phaseNumber:=8, act:=_off);
            fb_stopANU(phaseNumber:=9);
             fb_nu1Off(phaseNumber:=11, act:=_off);
             fb_nu2Off(phaseNumber:=12, act:=_off);
            fb_stopNU1(phaseNumber:=15, act:=_off);
            fb_stopNU2(phaseNumber:=16, act:=_off);
  onInit:=TRUE;
  END_IF;

      fb_puskOilSystem(StrPh:=puskOilSystem, alg:=algoritms.puskOilSystem);
        fb_algContinue(StrQ:=algContinue);
              fb_nuOff(StrPh:=nuOff);
             fb_dPmgAi(StrPh:=dPmgAi, ai:=ai.dPmaslo_gaz, less:=im.testdPmg_Ust_dPLow.Value);
             fb_dPmgDi(StrPh:=dPmgDi);
               fb_nuOn(StrPh:=nuOn);
            fb_noRezrv(StrPh:=noRezrv);
   fb_testUnsuccessful(StrPh:=testUnsuccessful);
          fb_BreakTest(StrPh:=BreakTest, timer:=AlgTimers.testdPmg_BreakTest);
             fb_pnsOff(StrPh:=pnsOff, Im:=Im.pns);
            fb_stopANU(StrPh:=stopANU);
             fb_nu1Off(StrPh:=nu1Off, Im:=Im.nu1);
             fb_nu2Off(StrPh:=nu2Off, Im:=Im.nu2);
            fb_stopNU1(StrPh:=stopNU1, Im:=Im.nu1);
            fb_stopNU2(StrPh:=stopNU2, Im:=Im.nu2);

  StrAlg.CanRun := StrAlg.inCanRun;
  StrAlg.OpcCommandsDisabled := StrAlg.inOpcCommandsDisabled;

  IF StrAlg.isRuning THEN

      StrAlg.hasError := pnsOff.error OR nu1Off.error OR nu2Off.error
      OR stopNU1.error OR stopNU2.error OR testUnsuccessful.error;

      IF puskOilSystem.top THEN
           IF NOT _resetQuestion THEN
           askQuestion(algContinue);
            _resetQuestion:=TRUE;
           END_IF;
      END_IF;

      IF algContinue.answer = _Answers.ANS_YES AND NOT nuOff.top THEN

          runPhase(nuOff);

          IF Im.nu1.onStatus = _statusDualInput.STATUS_ON THEN
  		runPhase(nu1Off);
          END_IF;

          IF Im.nu2.onStatus = _statusDualInput.STATUS_ON THEN
  		runPhase(nu2Off);
          END_IF;

          resetQuestion(algContinue);

      END_IF;

      IF nuOff.start AND NOT nuOff.top THEN
            runPhase(BreakTest);
  	nuOff.top:= Im.nu1.onStatus = _statusDualInput.STATUS_Off
                    AND Im.nu2.onStatus = _statusDualInput.STATUS_Off;
      END_IF;

      IF nuOff.top THEN

          runPhase(dPmgAi);
          runPhase(dPmgDi);
      END_IF;

      IF dPmgDi.start AND NOT dPmgDi.top THEN
          dPmgDi.top:=Im.SingleSignals.dP_oilgaz_low.q;
      END_IF;

      IF dPmgAi.top AND dPmgDi.top THEN
          runPhase(nuOn);
          runPhase(noRezrv);
      END_IF;

      IF noRezrv.start AND NOT noRezrv.top THEN
          noRezrv.top:=NotHasRezervNU;
      END_IF;

       IF nuOn.start AND (NOT WaitOnNU.Q) THEN
          WaitOnNU(IN:=Im.nu1.onStatus = _statusDualInput.STATUS_On OR
              Im.nu2.onStatus = _statusDualInput.STATUS_On, PT:=T#2S);
          nuOn.top:=Im.nu1.onStatus = _statusDualInput.STATUS_On OR
              Im.nu2.onStatus = _statusDualInput.STATUS_On;
      END_IF;

      IF  WaitOnNU.Q AND noRezrv.top THEN
          ai.dPmaslo_gaz.Disabled_LA:=TRUE;
          ai.dPmaslo_gaz.Disabled_LW:=TRUE;
          IM.SingleSignals.dP_oilgaz_low.Disabled_Sig:=TRUE;
          IM.SingleSignals.P_oil_low.Disabled_Sig:=TRUE;
          ai.P_masla_smazki_nizkoe.Disabled_LA:=TRUE;
          ai.P_masla_smazki_nizkoe.Disabled_LW:=TRUE;
          ai.P_masla_smazki_srednee_posle_nasosov.Disabled_LW:=TRUE;

          resetAiProtection(protections.P_masla_smazki_nizkoe_LA);
          resetDiProtection(protections.DavlenieMaslaSmazkiDi);
          resetAiProtection(protections.dP_maslogaz_LA);
          resetDiProtection(protections.dP_masloGaz_LowDI);

          resetIfRunning(algoritms.autoNu);
          resetIfRunning(algoritms.AutoPns);

          runPhase(stopANU);
          runPhase(pnsOff);

          runPhase(stopNU1);
          runPhase(stopNU2);

      END_IF;

      IF stopANU.start AND NOT stopANU.top THEN

  	stopANU.top:= Im.nu1.onStatus = _statusDualInput.STATUS_Off AND
                          Im.nu2.onStatus = _statusDualInput.STATUS_Off;
      END_IF;

      IF BreakTest.top AND NOT pnsOff.top THEN
  	testUnsuccessful.error:=TRUE;
      END_IF;

      IF pnsOff.top AND stopANU.top THEN
            resetPhase(BreakTest);
  	waitReset(IN:=TRUE, PT:= T#3S);
      END_IF;

      IF waitReset.Q THEN
          algManager.nMode:=ModeGpa.MODE_STOP;
          resetIfRunning(StrAlg);
      END_IF;

      StrAlg.isEnded:= pnsOff.top AND stopANU.top;

  END_IF;

  StrAlg.CanRun := StrAlg.inCanRun;
  StrAlg.OpcCommandsDisabled := StrAlg.inOpcCommandsDisabled;

  (* ---- Если управление с ВУ заблокировано, то  передаем команду из алгоритма ---- *)
  IF StrAlg.inOpcCommandsDisabled THEN
  	StrAlg.inCommand := StrAlg.inCommand_Alg;
  ELSE (* иначе передаем команду с АРМа*)
  	StrAlg.inCommand := StrAlg.inCommand_ARM;
  END_IF;

  _sunpackerCommand(command := StrAlg.inCommand);
  	source := _sunpackerCommand.source;
  	cmd := _sunpackerCommand.cmd;

  IF cmd <> 0 AND lastCmd <> cmd AND (((NOT StrAlg.opcCommandsDisabled) AND source > 0) OR source = 0) then
  	CASE BYTE_TO_INT(cmd) OF
  		(*cmdRun*) 1: 	IF (StrAlg.CanRun) THEN
  					StrAlg.isRuning := TRUE;
  					StrAlg.isEnded := FALSE;
  					StrAlg.hasError := FALSE;
  					(*****************       OnRun       *****************)

                                                    algManager.nMode:=ModeGpa.MODE_TESTDPMG;
                                                    resetAndDisable(alg:=algoritms.ppu);
                                                    algoritms.puskOilSystem.inCanRun:= TRUE;
                                                    runPhase(puskOilSystem);

  					cmd_for_Status := cmd;
  					source_for_Status := source;
  					command_error_for_Status := 0;
  				ELSE
  					StrAlg.isRuning := FALSE;
  					StrAlg.isEnded := FALSE;
  					StrAlg.hasError 	:= FALSE;

  					cmd_for_Status := 0;
  					source_for_Status := source;
  					command_error_for_Status := cmd;
  				END_IF;
  		(*cmdReset*) 2: 	StrAlg.isRuning := FALSE;
  				StrAlg.isEnded := FALSE;
  				StrAlg.hasError 	:= FALSE;

                                           (*****************       OnReset       *****************)
                                          waitReset(IN:=FALSE);
                                          WaitOnNU(IN:=FALSE);
                                          _resetQuestion:=FALSE;
                                          ai.P_masla_smazki_nizkoe.Disabled_LA:=TRUE;
                                          ai.P_masla_smazki_nizkoe.Disabled_LW:=TRUE;
                                          ai.P_masla_smazki_srednee_posle_nasosov.Disabled_LW:=TRUE;
                                          IM.SingleSignals.P_oil_low.Disabled_Sig:=TRUE;
                                          IM.SingleSignals.dP_oilgaz_low.Disabled_Sig:=TRUE;
                                          ai.dPmaslo_gaz.Disabled_LA:=TRUE;
                                          ai.dPmaslo_gaz.Disabled_LW:=TRUE;
                                          resetAiProtection(protections.P_masla_smazki_nizkoe_LA);
                                          resetDiProtection(protections.DavlenieMaslaSmazkiDi);
                                          resetAiProtection(protections.dP_maslogaz_LA);
                                          resetDiProtection(protections.dP_masloGaz_LowDI);

                                          resetPhase(puskOilSystem);
                                          resetPhase(nuOff);
                                          resetPhase(dPmgAi);
                                          resetPhase(dPmgDi);
                                          resetPhase(nuOn);
                                          resetPhase(noRezrv);
                                          resetPhase(BreakTest);
                                          resetPhase(testUnsuccessful);
                                          resetPhase(pnsOff);
                                          resetPhase(stopANU);
                                          resetPhase(nu1Off);
                                          resetPhase(nu2Off);
                                          resetPhase(stopNU1);
                                          resetPhase(stopNU2);

                                          resetQuestion(algContinue);
